(* PLC project PLC Using structs as arrays, CODESYS CODESYS V3.5 SP16, author Toni Kucic *)
(* stored: creationDateTime 2021-02-20T20:12:28.2562031, version 1.0, modificationDateTime 2021-02-20T20:12:09.3479166, organization TK Automation *)
(* A tutorial how to use structs and user derived types as arrays if the PLC IDE/Compiler doesnt allow for arrays. Working with booleans, numbers and user data types is shown in respective POUs that can be run on any PLC that is iec61131-3 compliant. For other data types the process is the same. On top of the examples the project contains struct arrays of 32 elements for each elementary type so the users can start using the functions immediately. If the operator needs different data types the Python generator script can be used. THe python script is located in the same repository as this file. Originally written in CODESYS 3.5. These DTs and POUs can be used under the MIT license. *)

TYPE BOOL32 : STRUCT
  ix00 : BOOL;  (* Index 00 of struct array *)
  ix01 : BOOL;  (* Index 01 of struct array *)
  ix02 : BOOL;  (* Index 02 of struct array *)
  ix03 : BOOL;  (* Index 03 of struct array *)
  ix04 : BOOL;  (* Index 04 of struct array *)
  ix05 : BOOL;  (* Index 05 of struct array *)
  ix06 : BOOL;  (* Index 06 of struct array *)
  ix07 : BOOL;  (* Index 07 of struct array *)
  ix08 : BOOL;  (* Index 08 of struct array *)
  ix09 : BOOL;  (* Index 09 of struct array *)
  ix10 : BOOL;  (* Index 10 of struct array *)
  ix11 : BOOL;  (* Index 11 of struct array *)
  ix12 : BOOL;  (* Index 12 of struct array *)
  ix13 : BOOL;  (* Index 13 of struct array *)
  ix14 : BOOL;  (* Index 14 of struct array *)
  ix15 : BOOL;  (* Index 15 of struct array *)
  ix16 : BOOL;  (* Index 16 of struct array *)
  ix17 : BOOL;  (* Index 17 of struct array *)
  ix18 : BOOL;  (* Index 18 of struct array *)
  ix19 : BOOL;  (* Index 19 of struct array *)
  ix20 : BOOL;  (* Index 20 of struct array *)
  ix21 : BOOL;  (* Index 21 of struct array *)
  ix22 : BOOL;  (* Index 22 of struct array *)
  ix23 : BOOL;  (* Index 23 of struct array *)
  ix24 : BOOL;  (* Index 24 of struct array *)
  ix25 : BOOL;  (* Index 25 of struct array *)
  ix26 : BOOL;  (* Index 26 of struct array *)
  ix27 : BOOL;  (* Index 27 of struct array *)
  ix28 : BOOL;  (* Index 28 of struct array *)
  ix29 : BOOL;  (* Index 29 of struct array *)
  ix30 : BOOL;  (* Index 30 of struct array *)
  ix31 : BOOL;  (* Index 31 of struct array *)
END_STRUCT;
END_TYPE

TYPE BYTE32 : STRUCT
  ix00 : BYTE;  (* Index 00 of struct array *)
  ix01 : BYTE;  (* Index 01 of struct array *)
  ix02 : BYTE;  (* Index 02 of struct array *)
  ix03 : BYTE;  (* Index 03 of struct array *)
  ix04 : BYTE;  (* Index 04 of struct array *)
  ix05 : BYTE;  (* Index 05 of struct array *)
  ix06 : BYTE;  (* Index 06 of struct array *)
  ix07 : BYTE;  (* Index 07 of struct array *)
  ix08 : BYTE;  (* Index 08 of struct array *)
  ix09 : BYTE;  (* Index 09 of struct array *)
  ix10 : BYTE;  (* Index 10 of struct array *)
  ix11 : BYTE;  (* Index 11 of struct array *)
  ix12 : BYTE;  (* Index 12 of struct array *)
  ix13 : BYTE;  (* Index 13 of struct array *)
  ix14 : BYTE;  (* Index 14 of struct array *)
  ix15 : BYTE;  (* Index 15 of struct array *)
  ix16 : BYTE;  (* Index 16 of struct array *)
  ix17 : BYTE;  (* Index 17 of struct array *)
  ix18 : BYTE;  (* Index 18 of struct array *)
  ix19 : BYTE;  (* Index 19 of struct array *)
  ix20 : BYTE;  (* Index 20 of struct array *)
  ix21 : BYTE;  (* Index 21 of struct array *)
  ix22 : BYTE;  (* Index 22 of struct array *)
  ix23 : BYTE;  (* Index 23 of struct array *)
  ix24 : BYTE;  (* Index 24 of struct array *)
  ix25 : BYTE;  (* Index 25 of struct array *)
  ix26 : BYTE;  (* Index 26 of struct array *)
  ix27 : BYTE;  (* Index 27 of struct array *)
  ix28 : BYTE;  (* Index 28 of struct array *)
  ix29 : BYTE;  (* Index 29 of struct array *)
  ix30 : BYTE;  (* Index 30 of struct array *)
  ix31 : BYTE;  (* Index 31 of struct array *)
END_STRUCT;
END_TYPE

TYPE DATE_AND_TIME32 : STRUCT
  ix00 : DT;  (* Index 00 of struct array *)
  ix01 : DT;  (* Index 01 of struct array *)
  ix02 : DT;  (* Index 02 of struct array *)
  ix03 : DT;  (* Index 03 of struct array *)
  ix04 : DT;  (* Index 04 of struct array *)
  ix05 : DT;  (* Index 05 of struct array *)
  ix06 : DT;  (* Index 06 of struct array *)
  ix07 : DT;  (* Index 07 of struct array *)
  ix08 : DT;  (* Index 08 of struct array *)
  ix09 : DT;  (* Index 09 of struct array *)
  ix10 : DT;  (* Index 10 of struct array *)
  ix11 : DT;  (* Index 11 of struct array *)
  ix12 : DT;  (* Index 12 of struct array *)
  ix13 : DT;  (* Index 13 of struct array *)
  ix14 : DT;  (* Index 14 of struct array *)
  ix15 : DT;  (* Index 15 of struct array *)
  ix16 : DT;  (* Index 16 of struct array *)
  ix17 : DT;  (* Index 17 of struct array *)
  ix18 : DT;  (* Index 18 of struct array *)
  ix19 : DT;  (* Index 19 of struct array *)
  ix20 : DT;  (* Index 20 of struct array *)
  ix21 : DT;  (* Index 21 of struct array *)
  ix22 : DT;  (* Index 22 of struct array *)
  ix23 : DT;  (* Index 23 of struct array *)
  ix24 : DT;  (* Index 24 of struct array *)
  ix25 : DT;  (* Index 25 of struct array *)
  ix26 : DT;  (* Index 26 of struct array *)
  ix27 : DT;  (* Index 27 of struct array *)
  ix28 : DT;  (* Index 28 of struct array *)
  ix29 : DT;  (* Index 29 of struct array *)
  ix30 : DT;  (* Index 30 of struct array *)
  ix31 : DT;  (* Index 31 of struct array *)
END_STRUCT;
END_TYPE

TYPE DATE32 : STRUCT
  ix00 : DATE;  (* Index 00 of struct array *)
  ix01 : DATE;  (* Index 01 of struct array *)
  ix02 : DATE;  (* Index 02 of struct array *)
  ix03 : DATE;  (* Index 03 of struct array *)
  ix04 : DATE;  (* Index 04 of struct array *)
  ix05 : DATE;  (* Index 05 of struct array *)
  ix06 : DATE;  (* Index 06 of struct array *)
  ix07 : DATE;  (* Index 07 of struct array *)
  ix08 : DATE;  (* Index 08 of struct array *)
  ix09 : DATE;  (* Index 09 of struct array *)
  ix10 : DATE;  (* Index 10 of struct array *)
  ix11 : DATE;  (* Index 11 of struct array *)
  ix12 : DATE;  (* Index 12 of struct array *)
  ix13 : DATE;  (* Index 13 of struct array *)
  ix14 : DATE;  (* Index 14 of struct array *)
  ix15 : DATE;  (* Index 15 of struct array *)
  ix16 : DATE;  (* Index 16 of struct array *)
  ix17 : DATE;  (* Index 17 of struct array *)
  ix18 : DATE;  (* Index 18 of struct array *)
  ix19 : DATE;  (* Index 19 of struct array *)
  ix20 : DATE;  (* Index 20 of struct array *)
  ix21 : DATE;  (* Index 21 of struct array *)
  ix22 : DATE;  (* Index 22 of struct array *)
  ix23 : DATE;  (* Index 23 of struct array *)
  ix24 : DATE;  (* Index 24 of struct array *)
  ix25 : DATE;  (* Index 25 of struct array *)
  ix26 : DATE;  (* Index 26 of struct array *)
  ix27 : DATE;  (* Index 27 of struct array *)
  ix28 : DATE;  (* Index 28 of struct array *)
  ix29 : DATE;  (* Index 29 of struct array *)
  ix30 : DATE;  (* Index 30 of struct array *)
  ix31 : DATE;  (* Index 31 of struct array *)
END_STRUCT;
END_TYPE

TYPE DINT32 : STRUCT
  ix00 : DINT;  (* Index 00 of struct array *)
  ix01 : DINT;  (* Index 01 of struct array *)
  ix02 : DINT;  (* Index 02 of struct array *)
  ix03 : DINT;  (* Index 03 of struct array *)
  ix04 : DINT;  (* Index 04 of struct array *)
  ix05 : DINT;  (* Index 05 of struct array *)
  ix06 : DINT;  (* Index 06 of struct array *)
  ix07 : DINT;  (* Index 07 of struct array *)
  ix08 : DINT;  (* Index 08 of struct array *)
  ix09 : DINT;  (* Index 09 of struct array *)
  ix10 : DINT;  (* Index 10 of struct array *)
  ix11 : DINT;  (* Index 11 of struct array *)
  ix12 : DINT;  (* Index 12 of struct array *)
  ix13 : DINT;  (* Index 13 of struct array *)
  ix14 : DINT;  (* Index 14 of struct array *)
  ix15 : DINT;  (* Index 15 of struct array *)
  ix16 : DINT;  (* Index 16 of struct array *)
  ix17 : DINT;  (* Index 17 of struct array *)
  ix18 : DINT;  (* Index 18 of struct array *)
  ix19 : DINT;  (* Index 19 of struct array *)
  ix20 : DINT;  (* Index 20 of struct array *)
  ix21 : DINT;  (* Index 21 of struct array *)
  ix22 : DINT;  (* Index 22 of struct array *)
  ix23 : DINT;  (* Index 23 of struct array *)
  ix24 : DINT;  (* Index 24 of struct array *)
  ix25 : DINT;  (* Index 25 of struct array *)
  ix26 : DINT;  (* Index 26 of struct array *)
  ix27 : DINT;  (* Index 27 of struct array *)
  ix28 : DINT;  (* Index 28 of struct array *)
  ix29 : DINT;  (* Index 29 of struct array *)
  ix30 : DINT;  (* Index 30 of struct array *)
  ix31 : DINT;  (* Index 31 of struct array *)
END_STRUCT;
END_TYPE

TYPE DWORD32 : STRUCT
  ix00 : DWORD;  (* Index 00 of struct array *)
  ix01 : DWORD;  (* Index 01 of struct array *)
  ix02 : DWORD;  (* Index 02 of struct array *)
  ix03 : DWORD;  (* Index 03 of struct array *)
  ix04 : DWORD;  (* Index 04 of struct array *)
  ix05 : DWORD;  (* Index 05 of struct array *)
  ix06 : DWORD;  (* Index 06 of struct array *)
  ix07 : DWORD;  (* Index 07 of struct array *)
  ix08 : DWORD;  (* Index 08 of struct array *)
  ix09 : DWORD;  (* Index 09 of struct array *)
  ix10 : DWORD;  (* Index 10 of struct array *)
  ix11 : DWORD;  (* Index 11 of struct array *)
  ix12 : DWORD;  (* Index 12 of struct array *)
  ix13 : DWORD;  (* Index 13 of struct array *)
  ix14 : DWORD;  (* Index 14 of struct array *)
  ix15 : DWORD;  (* Index 15 of struct array *)
  ix16 : DWORD;  (* Index 16 of struct array *)
  ix17 : DWORD;  (* Index 17 of struct array *)
  ix18 : DWORD;  (* Index 18 of struct array *)
  ix19 : DWORD;  (* Index 19 of struct array *)
  ix20 : DWORD;  (* Index 20 of struct array *)
  ix21 : DWORD;  (* Index 21 of struct array *)
  ix22 : DWORD;  (* Index 22 of struct array *)
  ix23 : DWORD;  (* Index 23 of struct array *)
  ix24 : DWORD;  (* Index 24 of struct array *)
  ix25 : DWORD;  (* Index 25 of struct array *)
  ix26 : DWORD;  (* Index 26 of struct array *)
  ix27 : DWORD;  (* Index 27 of struct array *)
  ix28 : DWORD;  (* Index 28 of struct array *)
  ix29 : DWORD;  (* Index 29 of struct array *)
  ix30 : DWORD;  (* Index 30 of struct array *)
  ix31 : DWORD;  (* Index 31 of struct array *)
END_STRUCT;
END_TYPE

TYPE INT32 : STRUCT
  ix00 : INT;  (* Index 00 of struct array *)
  ix01 : INT;  (* Index 01 of struct array *)
  ix02 : INT;  (* Index 02 of struct array *)
  ix03 : INT;  (* Index 03 of struct array *)
  ix04 : INT;  (* Index 04 of struct array *)
  ix05 : INT;  (* Index 05 of struct array *)
  ix06 : INT;  (* Index 06 of struct array *)
  ix07 : INT;  (* Index 07 of struct array *)
  ix08 : INT;  (* Index 08 of struct array *)
  ix09 : INT;  (* Index 09 of struct array *)
  ix10 : INT;  (* Index 10 of struct array *)
  ix11 : INT;  (* Index 11 of struct array *)
  ix12 : INT;  (* Index 12 of struct array *)
  ix13 : INT;  (* Index 13 of struct array *)
  ix14 : INT;  (* Index 14 of struct array *)
  ix15 : INT;  (* Index 15 of struct array *)
  ix16 : INT;  (* Index 16 of struct array *)
  ix17 : INT;  (* Index 17 of struct array *)
  ix18 : INT;  (* Index 18 of struct array *)
  ix19 : INT;  (* Index 19 of struct array *)
  ix20 : INT;  (* Index 20 of struct array *)
  ix21 : INT;  (* Index 21 of struct array *)
  ix22 : INT;  (* Index 22 of struct array *)
  ix23 : INT;  (* Index 23 of struct array *)
  ix24 : INT;  (* Index 24 of struct array *)
  ix25 : INT;  (* Index 25 of struct array *)
  ix26 : INT;  (* Index 26 of struct array *)
  ix27 : INT;  (* Index 27 of struct array *)
  ix28 : INT;  (* Index 28 of struct array *)
  ix29 : INT;  (* Index 29 of struct array *)
  ix30 : INT;  (* Index 30 of struct array *)
  ix31 : INT;  (* Index 31 of struct array *)
END_STRUCT;
END_TYPE

TYPE LDATE_AND_TIME32 : STRUCT
  ix00 : LDATE_AND_TIME;  (* Index 00 of struct array *)
  ix01 : LDATE_AND_TIME;  (* Index 01 of struct array *)
  ix02 : LDATE_AND_TIME;  (* Index 02 of struct array *)
  ix03 : LDATE_AND_TIME;  (* Index 03 of struct array *)
  ix04 : LDATE_AND_TIME;  (* Index 04 of struct array *)
  ix05 : LDATE_AND_TIME;  (* Index 05 of struct array *)
  ix06 : LDATE_AND_TIME;  (* Index 06 of struct array *)
  ix07 : LDATE_AND_TIME;  (* Index 07 of struct array *)
  ix08 : LDATE_AND_TIME;  (* Index 08 of struct array *)
  ix09 : LDATE_AND_TIME;  (* Index 09 of struct array *)
  ix10 : LDATE_AND_TIME;  (* Index 10 of struct array *)
  ix11 : LDATE_AND_TIME;  (* Index 11 of struct array *)
  ix12 : LDATE_AND_TIME;  (* Index 12 of struct array *)
  ix13 : LDATE_AND_TIME;  (* Index 13 of struct array *)
  ix14 : LDATE_AND_TIME;  (* Index 14 of struct array *)
  ix15 : LDATE_AND_TIME;  (* Index 15 of struct array *)
  ix16 : LDATE_AND_TIME;  (* Index 16 of struct array *)
  ix17 : LDATE_AND_TIME;  (* Index 17 of struct array *)
  ix18 : LDATE_AND_TIME;  (* Index 18 of struct array *)
  ix19 : LDATE_AND_TIME;  (* Index 19 of struct array *)
  ix20 : LDATE_AND_TIME;  (* Index 20 of struct array *)
  ix21 : LDATE_AND_TIME;  (* Index 21 of struct array *)
  ix22 : LDATE_AND_TIME;  (* Index 22 of struct array *)
  ix23 : LDATE_AND_TIME;  (* Index 23 of struct array *)
  ix24 : LDATE_AND_TIME;  (* Index 24 of struct array *)
  ix25 : LDATE_AND_TIME;  (* Index 25 of struct array *)
  ix26 : LDATE_AND_TIME;  (* Index 26 of struct array *)
  ix27 : LDATE_AND_TIME;  (* Index 27 of struct array *)
  ix28 : LDATE_AND_TIME;  (* Index 28 of struct array *)
  ix29 : LDATE_AND_TIME;  (* Index 29 of struct array *)
  ix30 : LDATE_AND_TIME;  (* Index 30 of struct array *)
  ix31 : LDATE_AND_TIME;  (* Index 31 of struct array *)
END_STRUCT;
END_TYPE

TYPE LDATE32 : STRUCT
  ix00 : LDATE;  (* Index 00 of struct array *)
  ix01 : LDATE;  (* Index 01 of struct array *)
  ix02 : LDATE;  (* Index 02 of struct array *)
  ix03 : LDATE;  (* Index 03 of struct array *)
  ix04 : LDATE;  (* Index 04 of struct array *)
  ix05 : LDATE;  (* Index 05 of struct array *)
  ix06 : LDATE;  (* Index 06 of struct array *)
  ix07 : LDATE;  (* Index 07 of struct array *)
  ix08 : LDATE;  (* Index 08 of struct array *)
  ix09 : LDATE;  (* Index 09 of struct array *)
  ix10 : LDATE;  (* Index 10 of struct array *)
  ix11 : LDATE;  (* Index 11 of struct array *)
  ix12 : LDATE;  (* Index 12 of struct array *)
  ix13 : LDATE;  (* Index 13 of struct array *)
  ix14 : LDATE;  (* Index 14 of struct array *)
  ix15 : LDATE;  (* Index 15 of struct array *)
  ix16 : LDATE;  (* Index 16 of struct array *)
  ix17 : LDATE;  (* Index 17 of struct array *)
  ix18 : LDATE;  (* Index 18 of struct array *)
  ix19 : LDATE;  (* Index 19 of struct array *)
  ix20 : LDATE;  (* Index 20 of struct array *)
  ix21 : LDATE;  (* Index 21 of struct array *)
  ix22 : LDATE;  (* Index 22 of struct array *)
  ix23 : LDATE;  (* Index 23 of struct array *)
  ix24 : LDATE;  (* Index 24 of struct array *)
  ix25 : LDATE;  (* Index 25 of struct array *)
  ix26 : LDATE;  (* Index 26 of struct array *)
  ix27 : LDATE;  (* Index 27 of struct array *)
  ix28 : LDATE;  (* Index 28 of struct array *)
  ix29 : LDATE;  (* Index 29 of struct array *)
  ix30 : LDATE;  (* Index 30 of struct array *)
  ix31 : LDATE;  (* Index 31 of struct array *)
END_STRUCT;
END_TYPE

TYPE LINT32 : STRUCT
  ix00 : LINT;  (* Index 00 of struct array *)
  ix01 : LINT;  (* Index 01 of struct array *)
  ix02 : LINT;  (* Index 02 of struct array *)
  ix03 : LINT;  (* Index 03 of struct array *)
  ix04 : LINT;  (* Index 04 of struct array *)
  ix05 : LINT;  (* Index 05 of struct array *)
  ix06 : LINT;  (* Index 06 of struct array *)
  ix07 : LINT;  (* Index 07 of struct array *)
  ix08 : LINT;  (* Index 08 of struct array *)
  ix09 : LINT;  (* Index 09 of struct array *)
  ix10 : LINT;  (* Index 10 of struct array *)
  ix11 : LINT;  (* Index 11 of struct array *)
  ix12 : LINT;  (* Index 12 of struct array *)
  ix13 : LINT;  (* Index 13 of struct array *)
  ix14 : LINT;  (* Index 14 of struct array *)
  ix15 : LINT;  (* Index 15 of struct array *)
  ix16 : LINT;  (* Index 16 of struct array *)
  ix17 : LINT;  (* Index 17 of struct array *)
  ix18 : LINT;  (* Index 18 of struct array *)
  ix19 : LINT;  (* Index 19 of struct array *)
  ix20 : LINT;  (* Index 20 of struct array *)
  ix21 : LINT;  (* Index 21 of struct array *)
  ix22 : LINT;  (* Index 22 of struct array *)
  ix23 : LINT;  (* Index 23 of struct array *)
  ix24 : LINT;  (* Index 24 of struct array *)
  ix25 : LINT;  (* Index 25 of struct array *)
  ix26 : LINT;  (* Index 26 of struct array *)
  ix27 : LINT;  (* Index 27 of struct array *)
  ix28 : LINT;  (* Index 28 of struct array *)
  ix29 : LINT;  (* Index 29 of struct array *)
  ix30 : LINT;  (* Index 30 of struct array *)
  ix31 : LINT;  (* Index 31 of struct array *)
END_STRUCT;
END_TYPE

TYPE LREAL32 : STRUCT
  ix00 : LREAL;  (* Index 00 of struct array *)
  ix01 : LREAL;  (* Index 01 of struct array *)
  ix02 : LREAL;  (* Index 02 of struct array *)
  ix03 : LREAL;  (* Index 03 of struct array *)
  ix04 : LREAL;  (* Index 04 of struct array *)
  ix05 : LREAL;  (* Index 05 of struct array *)
  ix06 : LREAL;  (* Index 06 of struct array *)
  ix07 : LREAL;  (* Index 07 of struct array *)
  ix08 : LREAL;  (* Index 08 of struct array *)
  ix09 : LREAL;  (* Index 09 of struct array *)
  ix10 : LREAL;  (* Index 10 of struct array *)
  ix11 : LREAL;  (* Index 11 of struct array *)
  ix12 : LREAL;  (* Index 12 of struct array *)
  ix13 : LREAL;  (* Index 13 of struct array *)
  ix14 : LREAL;  (* Index 14 of struct array *)
  ix15 : LREAL;  (* Index 15 of struct array *)
  ix16 : LREAL;  (* Index 16 of struct array *)
  ix17 : LREAL;  (* Index 17 of struct array *)
  ix18 : LREAL;  (* Index 18 of struct array *)
  ix19 : LREAL;  (* Index 19 of struct array *)
  ix20 : LREAL;  (* Index 20 of struct array *)
  ix21 : LREAL;  (* Index 21 of struct array *)
  ix22 : LREAL;  (* Index 22 of struct array *)
  ix23 : LREAL;  (* Index 23 of struct array *)
  ix24 : LREAL;  (* Index 24 of struct array *)
  ix25 : LREAL;  (* Index 25 of struct array *)
  ix26 : LREAL;  (* Index 26 of struct array *)
  ix27 : LREAL;  (* Index 27 of struct array *)
  ix28 : LREAL;  (* Index 28 of struct array *)
  ix29 : LREAL;  (* Index 29 of struct array *)
  ix30 : LREAL;  (* Index 30 of struct array *)
  ix31 : LREAL;  (* Index 31 of struct array *)
END_STRUCT;
END_TYPE

TYPE LTIME_OF_DAY32 : STRUCT
  ix00 : LTIME_OF_DAY;  (* Index 00 of struct array *)
  ix01 : LTIME_OF_DAY;  (* Index 01 of struct array *)
  ix02 : LTIME_OF_DAY;  (* Index 02 of struct array *)
  ix03 : LTIME_OF_DAY;  (* Index 03 of struct array *)
  ix04 : LTIME_OF_DAY;  (* Index 04 of struct array *)
  ix05 : LTIME_OF_DAY;  (* Index 05 of struct array *)
  ix06 : LTIME_OF_DAY;  (* Index 06 of struct array *)
  ix07 : LTIME_OF_DAY;  (* Index 07 of struct array *)
  ix08 : LTIME_OF_DAY;  (* Index 08 of struct array *)
  ix09 : LTIME_OF_DAY;  (* Index 09 of struct array *)
  ix10 : LTIME_OF_DAY;  (* Index 10 of struct array *)
  ix11 : LTIME_OF_DAY;  (* Index 11 of struct array *)
  ix12 : LTIME_OF_DAY;  (* Index 12 of struct array *)
  ix13 : LTIME_OF_DAY;  (* Index 13 of struct array *)
  ix14 : LTIME_OF_DAY;  (* Index 14 of struct array *)
  ix15 : LTIME_OF_DAY;  (* Index 15 of struct array *)
  ix16 : LTIME_OF_DAY;  (* Index 16 of struct array *)
  ix17 : LTIME_OF_DAY;  (* Index 17 of struct array *)
  ix18 : LTIME_OF_DAY;  (* Index 18 of struct array *)
  ix19 : LTIME_OF_DAY;  (* Index 19 of struct array *)
  ix20 : LTIME_OF_DAY;  (* Index 20 of struct array *)
  ix21 : LTIME_OF_DAY;  (* Index 21 of struct array *)
  ix22 : LTIME_OF_DAY;  (* Index 22 of struct array *)
  ix23 : LTIME_OF_DAY;  (* Index 23 of struct array *)
  ix24 : LTIME_OF_DAY;  (* Index 24 of struct array *)
  ix25 : LTIME_OF_DAY;  (* Index 25 of struct array *)
  ix26 : LTIME_OF_DAY;  (* Index 26 of struct array *)
  ix27 : LTIME_OF_DAY;  (* Index 27 of struct array *)
  ix28 : LTIME_OF_DAY;  (* Index 28 of struct array *)
  ix29 : LTIME_OF_DAY;  (* Index 29 of struct array *)
  ix30 : LTIME_OF_DAY;  (* Index 30 of struct array *)
  ix31 : LTIME_OF_DAY;  (* Index 31 of struct array *)
END_STRUCT;
END_TYPE

TYPE LTIME32 : STRUCT
  ix00 : LTIME;  (* Index 00 of struct array *)
  ix01 : LTIME;  (* Index 01 of struct array *)
  ix02 : LTIME;  (* Index 02 of struct array *)
  ix03 : LTIME;  (* Index 03 of struct array *)
  ix04 : LTIME;  (* Index 04 of struct array *)
  ix05 : LTIME;  (* Index 05 of struct array *)
  ix06 : LTIME;  (* Index 06 of struct array *)
  ix07 : LTIME;  (* Index 07 of struct array *)
  ix08 : LTIME;  (* Index 08 of struct array *)
  ix09 : LTIME;  (* Index 09 of struct array *)
  ix10 : LTIME;  (* Index 10 of struct array *)
  ix11 : LTIME;  (* Index 11 of struct array *)
  ix12 : LTIME;  (* Index 12 of struct array *)
  ix13 : LTIME;  (* Index 13 of struct array *)
  ix14 : LTIME;  (* Index 14 of struct array *)
  ix15 : LTIME;  (* Index 15 of struct array *)
  ix16 : LTIME;  (* Index 16 of struct array *)
  ix17 : LTIME;  (* Index 17 of struct array *)
  ix18 : LTIME;  (* Index 18 of struct array *)
  ix19 : LTIME;  (* Index 19 of struct array *)
  ix20 : LTIME;  (* Index 20 of struct array *)
  ix21 : LTIME;  (* Index 21 of struct array *)
  ix22 : LTIME;  (* Index 22 of struct array *)
  ix23 : LTIME;  (* Index 23 of struct array *)
  ix24 : LTIME;  (* Index 24 of struct array *)
  ix25 : LTIME;  (* Index 25 of struct array *)
  ix26 : LTIME;  (* Index 26 of struct array *)
  ix27 : LTIME;  (* Index 27 of struct array *)
  ix28 : LTIME;  (* Index 28 of struct array *)
  ix29 : LTIME;  (* Index 29 of struct array *)
  ix30 : LTIME;  (* Index 30 of struct array *)
  ix31 : LTIME;  (* Index 31 of struct array *)
END_STRUCT;
END_TYPE

TYPE LWORD32 : STRUCT
  ix00 : LWORD;  (* Index 00 of struct array *)
  ix01 : LWORD;  (* Index 01 of struct array *)
  ix02 : LWORD;  (* Index 02 of struct array *)
  ix03 : LWORD;  (* Index 03 of struct array *)
  ix04 : LWORD;  (* Index 04 of struct array *)
  ix05 : LWORD;  (* Index 05 of struct array *)
  ix06 : LWORD;  (* Index 06 of struct array *)
  ix07 : LWORD;  (* Index 07 of struct array *)
  ix08 : LWORD;  (* Index 08 of struct array *)
  ix09 : LWORD;  (* Index 09 of struct array *)
  ix10 : LWORD;  (* Index 10 of struct array *)
  ix11 : LWORD;  (* Index 11 of struct array *)
  ix12 : LWORD;  (* Index 12 of struct array *)
  ix13 : LWORD;  (* Index 13 of struct array *)
  ix14 : LWORD;  (* Index 14 of struct array *)
  ix15 : LWORD;  (* Index 15 of struct array *)
  ix16 : LWORD;  (* Index 16 of struct array *)
  ix17 : LWORD;  (* Index 17 of struct array *)
  ix18 : LWORD;  (* Index 18 of struct array *)
  ix19 : LWORD;  (* Index 19 of struct array *)
  ix20 : LWORD;  (* Index 20 of struct array *)
  ix21 : LWORD;  (* Index 21 of struct array *)
  ix22 : LWORD;  (* Index 22 of struct array *)
  ix23 : LWORD;  (* Index 23 of struct array *)
  ix24 : LWORD;  (* Index 24 of struct array *)
  ix25 : LWORD;  (* Index 25 of struct array *)
  ix26 : LWORD;  (* Index 26 of struct array *)
  ix27 : LWORD;  (* Index 27 of struct array *)
  ix28 : LWORD;  (* Index 28 of struct array *)
  ix29 : LWORD;  (* Index 29 of struct array *)
  ix30 : LWORD;  (* Index 30 of struct array *)
  ix31 : LWORD;  (* Index 31 of struct array *)
END_STRUCT;
END_TYPE

TYPE REAL32 : STRUCT
  ix00 : REAL;  (* Index 00 of struct array *)
  ix01 : REAL;  (* Index 01 of struct array *)
  ix02 : REAL;  (* Index 02 of struct array *)
  ix03 : REAL;  (* Index 03 of struct array *)
  ix04 : REAL;  (* Index 04 of struct array *)
  ix05 : REAL;  (* Index 05 of struct array *)
  ix06 : REAL;  (* Index 06 of struct array *)
  ix07 : REAL;  (* Index 07 of struct array *)
  ix08 : REAL;  (* Index 08 of struct array *)
  ix09 : REAL;  (* Index 09 of struct array *)
  ix10 : REAL;  (* Index 10 of struct array *)
  ix11 : REAL;  (* Index 11 of struct array *)
  ix12 : REAL;  (* Index 12 of struct array *)
  ix13 : REAL;  (* Index 13 of struct array *)
  ix14 : REAL;  (* Index 14 of struct array *)
  ix15 : REAL;  (* Index 15 of struct array *)
  ix16 : REAL;  (* Index 16 of struct array *)
  ix17 : REAL;  (* Index 17 of struct array *)
  ix18 : REAL;  (* Index 18 of struct array *)
  ix19 : REAL;  (* Index 19 of struct array *)
  ix20 : REAL;  (* Index 20 of struct array *)
  ix21 : REAL;  (* Index 21 of struct array *)
  ix22 : REAL;  (* Index 22 of struct array *)
  ix23 : REAL;  (* Index 23 of struct array *)
  ix24 : REAL;  (* Index 24 of struct array *)
  ix25 : REAL;  (* Index 25 of struct array *)
  ix26 : REAL;  (* Index 26 of struct array *)
  ix27 : REAL;  (* Index 27 of struct array *)
  ix28 : REAL;  (* Index 28 of struct array *)
  ix29 : REAL;  (* Index 29 of struct array *)
  ix30 : REAL;  (* Index 30 of struct array *)
  ix31 : REAL;  (* Index 31 of struct array *)
END_STRUCT;
END_TYPE

TYPE SINT32 : STRUCT
  ix00 : SINT;  (* Index 00 of struct array *)
  ix01 : SINT;  (* Index 01 of struct array *)
  ix02 : SINT;  (* Index 02 of struct array *)
  ix03 : SINT;  (* Index 03 of struct array *)
  ix04 : SINT;  (* Index 04 of struct array *)
  ix05 : SINT;  (* Index 05 of struct array *)
  ix06 : SINT;  (* Index 06 of struct array *)
  ix07 : SINT;  (* Index 07 of struct array *)
  ix08 : SINT;  (* Index 08 of struct array *)
  ix09 : SINT;  (* Index 09 of struct array *)
  ix10 : SINT;  (* Index 10 of struct array *)
  ix11 : SINT;  (* Index 11 of struct array *)
  ix12 : SINT;  (* Index 12 of struct array *)
  ix13 : SINT;  (* Index 13 of struct array *)
  ix14 : SINT;  (* Index 14 of struct array *)
  ix15 : SINT;  (* Index 15 of struct array *)
  ix16 : SINT;  (* Index 16 of struct array *)
  ix17 : SINT;  (* Index 17 of struct array *)
  ix18 : SINT;  (* Index 18 of struct array *)
  ix19 : SINT;  (* Index 19 of struct array *)
  ix20 : SINT;  (* Index 20 of struct array *)
  ix21 : SINT;  (* Index 21 of struct array *)
  ix22 : SINT;  (* Index 22 of struct array *)
  ix23 : SINT;  (* Index 23 of struct array *)
  ix24 : SINT;  (* Index 24 of struct array *)
  ix25 : SINT;  (* Index 25 of struct array *)
  ix26 : SINT;  (* Index 26 of struct array *)
  ix27 : SINT;  (* Index 27 of struct array *)
  ix28 : SINT;  (* Index 28 of struct array *)
  ix29 : SINT;  (* Index 29 of struct array *)
  ix30 : SINT;  (* Index 30 of struct array *)
  ix31 : SINT;  (* Index 31 of struct array *)
END_STRUCT;
END_TYPE

TYPE STRING32 : STRUCT
  ix00 : STRING;  (* Index 00 of struct array *)
  ix01 : STRING;  (* Index 01 of struct array *)
  ix02 : STRING;  (* Index 02 of struct array *)
  ix03 : STRING;  (* Index 03 of struct array *)
  ix04 : STRING;  (* Index 04 of struct array *)
  ix05 : STRING;  (* Index 05 of struct array *)
  ix06 : STRING;  (* Index 06 of struct array *)
  ix07 : STRING;  (* Index 07 of struct array *)
  ix08 : STRING;  (* Index 08 of struct array *)
  ix09 : STRING;  (* Index 09 of struct array *)
  ix10 : STRING;  (* Index 10 of struct array *)
  ix11 : STRING;  (* Index 11 of struct array *)
  ix12 : STRING;  (* Index 12 of struct array *)
  ix13 : STRING;  (* Index 13 of struct array *)
  ix14 : STRING;  (* Index 14 of struct array *)
  ix15 : STRING;  (* Index 15 of struct array *)
  ix16 : STRING;  (* Index 16 of struct array *)
  ix17 : STRING;  (* Index 17 of struct array *)
  ix18 : STRING;  (* Index 18 of struct array *)
  ix19 : STRING;  (* Index 19 of struct array *)
  ix20 : STRING;  (* Index 20 of struct array *)
  ix21 : STRING;  (* Index 21 of struct array *)
  ix22 : STRING;  (* Index 22 of struct array *)
  ix23 : STRING;  (* Index 23 of struct array *)
  ix24 : STRING;  (* Index 24 of struct array *)
  ix25 : STRING;  (* Index 25 of struct array *)
  ix26 : STRING;  (* Index 26 of struct array *)
  ix27 : STRING;  (* Index 27 of struct array *)
  ix28 : STRING;  (* Index 28 of struct array *)
  ix29 : STRING;  (* Index 29 of struct array *)
  ix30 : STRING;  (* Index 30 of struct array *)
  ix31 : STRING;  (* Index 31 of struct array *)
END_STRUCT;
END_TYPE

TYPE TIME_OF_DAY32 : STRUCT
  ix00 : TOD;  (* Index 00 of struct array *)
  ix01 : TOD;  (* Index 01 of struct array *)
  ix02 : TOD;  (* Index 02 of struct array *)
  ix03 : TOD;  (* Index 03 of struct array *)
  ix04 : TOD;  (* Index 04 of struct array *)
  ix05 : TOD;  (* Index 05 of struct array *)
  ix06 : TOD;  (* Index 06 of struct array *)
  ix07 : TOD;  (* Index 07 of struct array *)
  ix08 : TOD;  (* Index 08 of struct array *)
  ix09 : TOD;  (* Index 09 of struct array *)
  ix10 : TOD;  (* Index 10 of struct array *)
  ix11 : TOD;  (* Index 11 of struct array *)
  ix12 : TOD;  (* Index 12 of struct array *)
  ix13 : TOD;  (* Index 13 of struct array *)
  ix14 : TOD;  (* Index 14 of struct array *)
  ix15 : TOD;  (* Index 15 of struct array *)
  ix16 : TOD;  (* Index 16 of struct array *)
  ix17 : TOD;  (* Index 17 of struct array *)
  ix18 : TOD;  (* Index 18 of struct array *)
  ix19 : TOD;  (* Index 19 of struct array *)
  ix20 : TOD;  (* Index 20 of struct array *)
  ix21 : TOD;  (* Index 21 of struct array *)
  ix22 : TOD;  (* Index 22 of struct array *)
  ix23 : TOD;  (* Index 23 of struct array *)
  ix24 : TOD;  (* Index 24 of struct array *)
  ix25 : TOD;  (* Index 25 of struct array *)
  ix26 : TOD;  (* Index 26 of struct array *)
  ix27 : TOD;  (* Index 27 of struct array *)
  ix28 : TOD;  (* Index 28 of struct array *)
  ix29 : TOD;  (* Index 29 of struct array *)
  ix30 : TOD;  (* Index 30 of struct array *)
  ix31 : TOD;  (* Index 31 of struct array *)
END_STRUCT;
END_TYPE

TYPE TIME32 : STRUCT
  ix00 : TIME;  (* Index 00 of struct array *)
  ix01 : TIME;  (* Index 01 of struct array *)
  ix02 : TIME;  (* Index 02 of struct array *)
  ix03 : TIME;  (* Index 03 of struct array *)
  ix04 : TIME;  (* Index 04 of struct array *)
  ix05 : TIME;  (* Index 05 of struct array *)
  ix06 : TIME;  (* Index 06 of struct array *)
  ix07 : TIME;  (* Index 07 of struct array *)
  ix08 : TIME;  (* Index 08 of struct array *)
  ix09 : TIME;  (* Index 09 of struct array *)
  ix10 : TIME;  (* Index 10 of struct array *)
  ix11 : TIME;  (* Index 11 of struct array *)
  ix12 : TIME;  (* Index 12 of struct array *)
  ix13 : TIME;  (* Index 13 of struct array *)
  ix14 : TIME;  (* Index 14 of struct array *)
  ix15 : TIME;  (* Index 15 of struct array *)
  ix16 : TIME;  (* Index 16 of struct array *)
  ix17 : TIME;  (* Index 17 of struct array *)
  ix18 : TIME;  (* Index 18 of struct array *)
  ix19 : TIME;  (* Index 19 of struct array *)
  ix20 : TIME;  (* Index 20 of struct array *)
  ix21 : TIME;  (* Index 21 of struct array *)
  ix22 : TIME;  (* Index 22 of struct array *)
  ix23 : TIME;  (* Index 23 of struct array *)
  ix24 : TIME;  (* Index 24 of struct array *)
  ix25 : TIME;  (* Index 25 of struct array *)
  ix26 : TIME;  (* Index 26 of struct array *)
  ix27 : TIME;  (* Index 27 of struct array *)
  ix28 : TIME;  (* Index 28 of struct array *)
  ix29 : TIME;  (* Index 29 of struct array *)
  ix30 : TIME;  (* Index 30 of struct array *)
  ix31 : TIME;  (* Index 31 of struct array *)
END_STRUCT;
END_TYPE

TYPE UDINT32 : STRUCT
  ix00 : UDINT;  (* Index 00 of struct array *)
  ix01 : UDINT;  (* Index 01 of struct array *)
  ix02 : UDINT;  (* Index 02 of struct array *)
  ix03 : UDINT;  (* Index 03 of struct array *)
  ix04 : UDINT;  (* Index 04 of struct array *)
  ix05 : UDINT;  (* Index 05 of struct array *)
  ix06 : UDINT;  (* Index 06 of struct array *)
  ix07 : UDINT;  (* Index 07 of struct array *)
  ix08 : UDINT;  (* Index 08 of struct array *)
  ix09 : UDINT;  (* Index 09 of struct array *)
  ix10 : UDINT;  (* Index 10 of struct array *)
  ix11 : UDINT;  (* Index 11 of struct array *)
  ix12 : UDINT;  (* Index 12 of struct array *)
  ix13 : UDINT;  (* Index 13 of struct array *)
  ix14 : UDINT;  (* Index 14 of struct array *)
  ix15 : UDINT;  (* Index 15 of struct array *)
  ix16 : UDINT;  (* Index 16 of struct array *)
  ix17 : UDINT;  (* Index 17 of struct array *)
  ix18 : UDINT;  (* Index 18 of struct array *)
  ix19 : UDINT;  (* Index 19 of struct array *)
  ix20 : UDINT;  (* Index 20 of struct array *)
  ix21 : UDINT;  (* Index 21 of struct array *)
  ix22 : UDINT;  (* Index 22 of struct array *)
  ix23 : UDINT;  (* Index 23 of struct array *)
  ix24 : UDINT;  (* Index 24 of struct array *)
  ix25 : UDINT;  (* Index 25 of struct array *)
  ix26 : UDINT;  (* Index 26 of struct array *)
  ix27 : UDINT;  (* Index 27 of struct array *)
  ix28 : UDINT;  (* Index 28 of struct array *)
  ix29 : UDINT;  (* Index 29 of struct array *)
  ix30 : UDINT;  (* Index 30 of struct array *)
  ix31 : UDINT;  (* Index 31 of struct array *)
END_STRUCT;
END_TYPE

TYPE UDT_Cmd : STRUCT
  StartCmd : BOOL;  (* Start command to the device *)
  StopCmd : BOOL;  (* Stop command to the device *)
  ResetCmd : BOOL;  (* Reset command for the device *)
  Ref : REAL;  (* Reference for the device to follow *)
END_STRUCT;
END_TYPE

TYPE UDT_Cmd32 : STRUCT
  udt00 : UDT_Cmd;  (* User data type array index 0 *)
  udt01 : UDT_Cmd;  (* User data type array index 1 *)
  udt02 : UDT_Cmd;  (* User data type array index 2 *)
  udt03 : UDT_Cmd;  (* User data type array index 3 *)
  udt04 : UDT_Cmd;  (* User data type array index 4 *)
  udt05 : UDT_Cmd;  (* User data type array index 5 *)
  udt06 : UDT_Cmd;  (* User data type array index 6 *)
  udt07 : UDT_Cmd;  (* User data type array index 7 *)
  udt08 : UDT_Cmd;  (* User data type array index 8 *)
  udt09 : UDT_Cmd;  (* User data type array index 9 *)
  udt10 : UDT_Cmd;  (* User data type array index 10 *)
  udt11 : UDT_Cmd;  (* User data type array index 11 *)
  udt12 : UDT_Cmd;  (* User data type array index 12 *)
  udt13 : UDT_Cmd;  (* User data type array index 13 *)
  udt14 : UDT_Cmd;  (* User data type array index 14 *)
  udt15 : UDT_Cmd;  (* User data type array index 15 *)
  udt16 : UDT_Cmd;  (* User data type array index 16 *)
  udt17 : UDT_Cmd;  (* User data type array index 17 *)
  udt18 : UDT_Cmd;  (* User data type array index 18 *)
  udt19 : UDT_Cmd;  (* User data type array index 19 *)
  udt20 : UDT_Cmd;  (* User data type array index 20 *)
  udt21 : UDT_Cmd;  (* User data type array index 21 *)
  udt22 : UDT_Cmd;  (* User data type array index 22 *)
  udt23 : UDT_Cmd;  (* User data type array index 23 *)
  udt24 : UDT_Cmd;  (* User data type array index 24 *)
  udt25 : UDT_Cmd;  (* User data type array index 25 *)
  udt26 : UDT_Cmd;  (* User data type array index 26 *)
  udt27 : UDT_Cmd;  (* User data type array index 27 *)
  udt28 : UDT_Cmd;  (* User data type array index 28 *)
  udt29 : UDT_Cmd;  (* User data type array index 29 *)
  udt30 : UDT_Cmd;  (* User data type array index 30 *)
  udt31 : UDT_Cmd;  (* User data type array index 31 *)
END_STRUCT;
END_TYPE

TYPE UDT_Status : STRUCT
  Running : BOOL;  (* Device is running *)
  ResetRequired : BOOL;  (* Device needs a reset *)
  RefActual : REAL;  (* Devices used reference *)
END_STRUCT;
END_TYPE

TYPE UDT_Status32 : STRUCT
  udt00 : UDT_Status;  (* User data type array index 0 *)
  udt01 : UDT_Status;  (* User data type array index 1 *)
  udt02 : UDT_Status;  (* User data type array index 2 *)
  udt03 : UDT_Status;  (* User data type array index 3 *)
  udt04 : UDT_Status;  (* User data type array index 4 *)
  udt05 : UDT_Status;  (* User data type array index 5 *)
  udt06 : UDT_Status;  (* User data type array index 6 *)
  udt07 : UDT_Status;  (* User data type array index 7 *)
  udt08 : UDT_Status;  (* User data type array index 8 *)
  udt09 : UDT_Status;  (* User data type array index 9 *)
  udt10 : UDT_Status;  (* User data type array index 10 *)
  udt11 : UDT_Status;  (* User data type array index 11 *)
  udt12 : UDT_Status;  (* User data type array index 12 *)
  udt13 : UDT_Status;  (* User data type array index 13 *)
  udt14 : UDT_Status;  (* User data type array index 14 *)
  udt15 : UDT_Status;  (* User data type array index 15 *)
  udt16 : UDT_Status;  (* User data type array index 16 *)
  udt17 : UDT_Status;  (* User data type array index 17 *)
  udt18 : UDT_Status;  (* User data type array index 18 *)
  udt19 : UDT_Status;  (* User data type array index 19 *)
  udt20 : UDT_Status;  (* User data type array index 20 *)
  udt21 : UDT_Status;  (* User data type array index 21 *)
  udt22 : UDT_Status;  (* User data type array index 22 *)
  udt23 : UDT_Status;  (* User data type array index 23 *)
  udt24 : UDT_Status;  (* User data type array index 24 *)
  udt25 : UDT_Status;  (* User data type array index 25 *)
  udt26 : UDT_Status;  (* User data type array index 26 *)
  udt27 : UDT_Status;  (* User data type array index 27 *)
  udt28 : UDT_Status;  (* User data type array index 28 *)
  udt29 : UDT_Status;  (* User data type array index 29 *)
  udt30 : UDT_Status;  (* User data type array index 30 *)
  udt31 : UDT_Status;  (* User data type array index 31 *)
END_STRUCT;
END_TYPE

TYPE UINT32 : STRUCT
  ix00 : UINT;  (* Index 00 of struct array *)
  ix01 : UINT;  (* Index 01 of struct array *)
  ix02 : UINT;  (* Index 02 of struct array *)
  ix03 : UINT;  (* Index 03 of struct array *)
  ix04 : UINT;  (* Index 04 of struct array *)
  ix05 : UINT;  (* Index 05 of struct array *)
  ix06 : UINT;  (* Index 06 of struct array *)
  ix07 : UINT;  (* Index 07 of struct array *)
  ix08 : UINT;  (* Index 08 of struct array *)
  ix09 : UINT;  (* Index 09 of struct array *)
  ix10 : UINT;  (* Index 10 of struct array *)
  ix11 : UINT;  (* Index 11 of struct array *)
  ix12 : UINT;  (* Index 12 of struct array *)
  ix13 : UINT;  (* Index 13 of struct array *)
  ix14 : UINT;  (* Index 14 of struct array *)
  ix15 : UINT;  (* Index 15 of struct array *)
  ix16 : UINT;  (* Index 16 of struct array *)
  ix17 : UINT;  (* Index 17 of struct array *)
  ix18 : UINT;  (* Index 18 of struct array *)
  ix19 : UINT;  (* Index 19 of struct array *)
  ix20 : UINT;  (* Index 20 of struct array *)
  ix21 : UINT;  (* Index 21 of struct array *)
  ix22 : UINT;  (* Index 22 of struct array *)
  ix23 : UINT;  (* Index 23 of struct array *)
  ix24 : UINT;  (* Index 24 of struct array *)
  ix25 : UINT;  (* Index 25 of struct array *)
  ix26 : UINT;  (* Index 26 of struct array *)
  ix27 : UINT;  (* Index 27 of struct array *)
  ix28 : UINT;  (* Index 28 of struct array *)
  ix29 : UINT;  (* Index 29 of struct array *)
  ix30 : UINT;  (* Index 30 of struct array *)
  ix31 : UINT;  (* Index 31 of struct array *)
END_STRUCT;
END_TYPE

TYPE ULINT32 : STRUCT
  ix00 : ULINT;  (* Index 00 of struct array *)
  ix01 : ULINT;  (* Index 01 of struct array *)
  ix02 : ULINT;  (* Index 02 of struct array *)
  ix03 : ULINT;  (* Index 03 of struct array *)
  ix04 : ULINT;  (* Index 04 of struct array *)
  ix05 : ULINT;  (* Index 05 of struct array *)
  ix06 : ULINT;  (* Index 06 of struct array *)
  ix07 : ULINT;  (* Index 07 of struct array *)
  ix08 : ULINT;  (* Index 08 of struct array *)
  ix09 : ULINT;  (* Index 09 of struct array *)
  ix10 : ULINT;  (* Index 10 of struct array *)
  ix11 : ULINT;  (* Index 11 of struct array *)
  ix12 : ULINT;  (* Index 12 of struct array *)
  ix13 : ULINT;  (* Index 13 of struct array *)
  ix14 : ULINT;  (* Index 14 of struct array *)
  ix15 : ULINT;  (* Index 15 of struct array *)
  ix16 : ULINT;  (* Index 16 of struct array *)
  ix17 : ULINT;  (* Index 17 of struct array *)
  ix18 : ULINT;  (* Index 18 of struct array *)
  ix19 : ULINT;  (* Index 19 of struct array *)
  ix20 : ULINT;  (* Index 20 of struct array *)
  ix21 : ULINT;  (* Index 21 of struct array *)
  ix22 : ULINT;  (* Index 22 of struct array *)
  ix23 : ULINT;  (* Index 23 of struct array *)
  ix24 : ULINT;  (* Index 24 of struct array *)
  ix25 : ULINT;  (* Index 25 of struct array *)
  ix26 : ULINT;  (* Index 26 of struct array *)
  ix27 : ULINT;  (* Index 27 of struct array *)
  ix28 : ULINT;  (* Index 28 of struct array *)
  ix29 : ULINT;  (* Index 29 of struct array *)
  ix30 : ULINT;  (* Index 30 of struct array *)
  ix31 : ULINT;  (* Index 31 of struct array *)
END_STRUCT;
END_TYPE

TYPE USINT32 : STRUCT
  ix00 : USINT;  (* Index 00 of struct array *)
  ix01 : USINT;  (* Index 01 of struct array *)
  ix02 : USINT;  (* Index 02 of struct array *)
  ix03 : USINT;  (* Index 03 of struct array *)
  ix04 : USINT;  (* Index 04 of struct array *)
  ix05 : USINT;  (* Index 05 of struct array *)
  ix06 : USINT;  (* Index 06 of struct array *)
  ix07 : USINT;  (* Index 07 of struct array *)
  ix08 : USINT;  (* Index 08 of struct array *)
  ix09 : USINT;  (* Index 09 of struct array *)
  ix10 : USINT;  (* Index 10 of struct array *)
  ix11 : USINT;  (* Index 11 of struct array *)
  ix12 : USINT;  (* Index 12 of struct array *)
  ix13 : USINT;  (* Index 13 of struct array *)
  ix14 : USINT;  (* Index 14 of struct array *)
  ix15 : USINT;  (* Index 15 of struct array *)
  ix16 : USINT;  (* Index 16 of struct array *)
  ix17 : USINT;  (* Index 17 of struct array *)
  ix18 : USINT;  (* Index 18 of struct array *)
  ix19 : USINT;  (* Index 19 of struct array *)
  ix20 : USINT;  (* Index 20 of struct array *)
  ix21 : USINT;  (* Index 21 of struct array *)
  ix22 : USINT;  (* Index 22 of struct array *)
  ix23 : USINT;  (* Index 23 of struct array *)
  ix24 : USINT;  (* Index 24 of struct array *)
  ix25 : USINT;  (* Index 25 of struct array *)
  ix26 : USINT;  (* Index 26 of struct array *)
  ix27 : USINT;  (* Index 27 of struct array *)
  ix28 : USINT;  (* Index 28 of struct array *)
  ix29 : USINT;  (* Index 29 of struct array *)
  ix30 : USINT;  (* Index 30 of struct array *)
  ix31 : USINT;  (* Index 31 of struct array *)
END_STRUCT;
END_TYPE

TYPE WORD32 : STRUCT
  ix00 : WORD;  (* Index 00 of struct array *)
  ix01 : WORD;  (* Index 01 of struct array *)
  ix02 : WORD;  (* Index 02 of struct array *)
  ix03 : WORD;  (* Index 03 of struct array *)
  ix04 : WORD;  (* Index 04 of struct array *)
  ix05 : WORD;  (* Index 05 of struct array *)
  ix06 : WORD;  (* Index 06 of struct array *)
  ix07 : WORD;  (* Index 07 of struct array *)
  ix08 : WORD;  (* Index 08 of struct array *)
  ix09 : WORD;  (* Index 09 of struct array *)
  ix10 : WORD;  (* Index 10 of struct array *)
  ix11 : WORD;  (* Index 11 of struct array *)
  ix12 : WORD;  (* Index 12 of struct array *)
  ix13 : WORD;  (* Index 13 of struct array *)
  ix14 : WORD;  (* Index 14 of struct array *)
  ix15 : WORD;  (* Index 15 of struct array *)
  ix16 : WORD;  (* Index 16 of struct array *)
  ix17 : WORD;  (* Index 17 of struct array *)
  ix18 : WORD;  (* Index 18 of struct array *)
  ix19 : WORD;  (* Index 19 of struct array *)
  ix20 : WORD;  (* Index 20 of struct array *)
  ix21 : WORD;  (* Index 21 of struct array *)
  ix22 : WORD;  (* Index 22 of struct array *)
  ix23 : WORD;  (* Index 23 of struct array *)
  ix24 : WORD;  (* Index 24 of struct array *)
  ix25 : WORD;  (* Index 25 of struct array *)
  ix26 : WORD;  (* Index 26 of struct array *)
  ix27 : WORD;  (* Index 27 of struct array *)
  ix28 : WORD;  (* Index 28 of struct array *)
  ix29 : WORD;  (* Index 29 of struct array *)
  ix30 : WORD;  (* Index 30 of struct array *)
  ix31 : WORD;  (* Index 31 of struct array *)
END_STRUCT;
END_TYPE

TYPE WSTRING32 : STRUCT
  ix00 : WSTRING;  (* Index 00 of struct array *)
  ix01 : WSTRING;  (* Index 01 of struct array *)
  ix02 : WSTRING;  (* Index 02 of struct array *)
  ix03 : WSTRING;  (* Index 03 of struct array *)
  ix04 : WSTRING;  (* Index 04 of struct array *)
  ix05 : WSTRING;  (* Index 05 of struct array *)
  ix06 : WSTRING;  (* Index 06 of struct array *)
  ix07 : WSTRING;  (* Index 07 of struct array *)
  ix08 : WSTRING;  (* Index 08 of struct array *)
  ix09 : WSTRING;  (* Index 09 of struct array *)
  ix10 : WSTRING;  (* Index 10 of struct array *)
  ix11 : WSTRING;  (* Index 11 of struct array *)
  ix12 : WSTRING;  (* Index 12 of struct array *)
  ix13 : WSTRING;  (* Index 13 of struct array *)
  ix14 : WSTRING;  (* Index 14 of struct array *)
  ix15 : WSTRING;  (* Index 15 of struct array *)
  ix16 : WSTRING;  (* Index 16 of struct array *)
  ix17 : WSTRING;  (* Index 17 of struct array *)
  ix18 : WSTRING;  (* Index 18 of struct array *)
  ix19 : WSTRING;  (* Index 19 of struct array *)
  ix20 : WSTRING;  (* Index 20 of struct array *)
  ix21 : WSTRING;  (* Index 21 of struct array *)
  ix22 : WSTRING;  (* Index 22 of struct array *)
  ix23 : WSTRING;  (* Index 23 of struct array *)
  ix24 : WSTRING;  (* Index 24 of struct array *)
  ix25 : WSTRING;  (* Index 25 of struct array *)
  ix26 : WSTRING;  (* Index 26 of struct array *)
  ix27 : WSTRING;  (* Index 27 of struct array *)
  ix28 : WSTRING;  (* Index 28 of struct array *)
  ix29 : WSTRING;  (* Index 29 of struct array *)
  ix30 : WSTRING;  (* Index 30 of struct array *)
  ix31 : WSTRING;  (* Index 31 of struct array *)
END_STRUCT;
END_TYPE

FUNCTION getBool32 : BOOL
  VAR_INPUT
    data : BOOL32;  (* Data to work on *)
    ix : USINT;  (* Index to retrieve *)
  END_VAR

            CASE ix OF
	0: getBool32 := data.ix00; (*Return index 0 for the data struct*)
	1: getBool32 := data.ix01; (*Return index 1 for the data struct*)
	2: getBool32 := data.ix02; (*Return index 2 for the data struct*)
	3: getBool32 := data.ix03; (*Return index 3 for the data struct*)
	4: getBool32 := data.ix04; (*Return index 4 for the data struct*)
	5: getBool32 := data.ix05; (*Return index 5 for the data struct*)
	6: getBool32 := data.ix06; (*Return index 6 for the data struct*)
	7: getBool32 := data.ix07; (*Return index 7 for the data struct*)
	8: getBool32 := data.ix08; (*Return index 8 for the data struct*)
	9: getBool32 := data.ix09; (*Return index 9 for the data struct*)
	10: getBool32 := data.ix10; (*Return index 10 for the data struct*)
	11: getBool32 := data.ix11; (*Return index 11 for the data struct*)
	12: getBool32 := data.ix12; (*Return index 12 for the data struct*)
	13: getBool32 := data.ix13; (*Return index 13 for the data struct*)
	14: getBool32 := data.ix14; (*Return index 14 for the data struct*)
	15: getBool32 := data.ix15; (*Return index 15 for the data struct*)
	16: getBool32 := data.ix16; (*Return index 16 for the data struct*)
	17: getBool32 := data.ix17; (*Return index 17 for the data struct*)
	18: getBool32 := data.ix18; (*Return index 18 for the data struct*)
	19: getBool32 := data.ix19; (*Return index 19 for the data struct*)
	20: getBool32 := data.ix20; (*Return index 20 for the data struct*)
	21: getBool32 := data.ix21; (*Return index 21 for the data struct*)
	22: getBool32 := data.ix22; (*Return index 22 for the data struct*)
	23: getBool32 := data.ix23; (*Return index 23 for the data struct*)
	24: getBool32 := data.ix24; (*Return index 24 for the data struct*)
	25: getBool32 := data.ix25; (*Return index 25 for the data struct*)
	26: getBool32 := data.ix26; (*Return index 26 for the data struct*)
	27: getBool32 := data.ix27; (*Return index 27 for the data struct*)
	28: getBool32 := data.ix28; (*Return index 28 for the data struct*)
	29: getBool32 := data.ix29; (*Return index 29 for the data struct*)
	30: getBool32 := data.ix30; (*Return index 30 for the data struct*)
	31: getBool32 := data.ix31; (*Return index 31 for the data struct*)
ELSE
	(*Index is invalid, return initial function value*)
	RETURN;
END_CASE
RETURN;

          
END_FUNCTION

FUNCTION getByte32 : BYTE
  VAR_INPUT
    data : BYTE32;  (* Data to work on *)
    ix : USINT;  (* Index to retrieve *)
  END_VAR

            CASE ix OF
	0: getByte32 := data.ix00; (*Return index 0 for the data struct*)
	1: getByte32 := data.ix01; (*Return index 1 for the data struct*)
	2: getByte32 := data.ix02; (*Return index 2 for the data struct*)
	3: getByte32 := data.ix03; (*Return index 3 for the data struct*)
	4: getByte32 := data.ix04; (*Return index 4 for the data struct*)
	5: getByte32 := data.ix05; (*Return index 5 for the data struct*)
	6: getByte32 := data.ix06; (*Return index 6 for the data struct*)
	7: getByte32 := data.ix07; (*Return index 7 for the data struct*)
	8: getByte32 := data.ix08; (*Return index 8 for the data struct*)
	9: getByte32 := data.ix09; (*Return index 9 for the data struct*)
	10: getByte32 := data.ix10; (*Return index 10 for the data struct*)
	11: getByte32 := data.ix11; (*Return index 11 for the data struct*)
	12: getByte32 := data.ix12; (*Return index 12 for the data struct*)
	13: getByte32 := data.ix13; (*Return index 13 for the data struct*)
	14: getByte32 := data.ix14; (*Return index 14 for the data struct*)
	15: getByte32 := data.ix15; (*Return index 15 for the data struct*)
	16: getByte32 := data.ix16; (*Return index 16 for the data struct*)
	17: getByte32 := data.ix17; (*Return index 17 for the data struct*)
	18: getByte32 := data.ix18; (*Return index 18 for the data struct*)
	19: getByte32 := data.ix19; (*Return index 19 for the data struct*)
	20: getByte32 := data.ix20; (*Return index 20 for the data struct*)
	21: getByte32 := data.ix21; (*Return index 21 for the data struct*)
	22: getByte32 := data.ix22; (*Return index 22 for the data struct*)
	23: getByte32 := data.ix23; (*Return index 23 for the data struct*)
	24: getByte32 := data.ix24; (*Return index 24 for the data struct*)
	25: getByte32 := data.ix25; (*Return index 25 for the data struct*)
	26: getByte32 := data.ix26; (*Return index 26 for the data struct*)
	27: getByte32 := data.ix27; (*Return index 27 for the data struct*)
	28: getByte32 := data.ix28; (*Return index 28 for the data struct*)
	29: getByte32 := data.ix29; (*Return index 29 for the data struct*)
	30: getByte32 := data.ix30; (*Return index 30 for the data struct*)
	31: getByte32 := data.ix31; (*Return index 31 for the data struct*)
ELSE
	(*Index is invalid, return initial function value*)
	RETURN;
END_CASE
RETURN;

          
END_FUNCTION

FUNCTION getDate_and_time32 : DT
  VAR_INPUT
    data : DATE_AND_TIME32;  (* Data to work on *)
    ix : USINT;  (* Index to retrieve *)
  END_VAR

            CASE ix OF
	0: getDate_and_time32 := data.ix00; (*Return index 0 for the data struct*)
	1: getDate_and_time32 := data.ix01; (*Return index 1 for the data struct*)
	2: getDate_and_time32 := data.ix02; (*Return index 2 for the data struct*)
	3: getDate_and_time32 := data.ix03; (*Return index 3 for the data struct*)
	4: getDate_and_time32 := data.ix04; (*Return index 4 for the data struct*)
	5: getDate_and_time32 := data.ix05; (*Return index 5 for the data struct*)
	6: getDate_and_time32 := data.ix06; (*Return index 6 for the data struct*)
	7: getDate_and_time32 := data.ix07; (*Return index 7 for the data struct*)
	8: getDate_and_time32 := data.ix08; (*Return index 8 for the data struct*)
	9: getDate_and_time32 := data.ix09; (*Return index 9 for the data struct*)
	10: getDate_and_time32 := data.ix10; (*Return index 10 for the data struct*)
	11: getDate_and_time32 := data.ix11; (*Return index 11 for the data struct*)
	12: getDate_and_time32 := data.ix12; (*Return index 12 for the data struct*)
	13: getDate_and_time32 := data.ix13; (*Return index 13 for the data struct*)
	14: getDate_and_time32 := data.ix14; (*Return index 14 for the data struct*)
	15: getDate_and_time32 := data.ix15; (*Return index 15 for the data struct*)
	16: getDate_and_time32 := data.ix16; (*Return index 16 for the data struct*)
	17: getDate_and_time32 := data.ix17; (*Return index 17 for the data struct*)
	18: getDate_and_time32 := data.ix18; (*Return index 18 for the data struct*)
	19: getDate_and_time32 := data.ix19; (*Return index 19 for the data struct*)
	20: getDate_and_time32 := data.ix20; (*Return index 20 for the data struct*)
	21: getDate_and_time32 := data.ix21; (*Return index 21 for the data struct*)
	22: getDate_and_time32 := data.ix22; (*Return index 22 for the data struct*)
	23: getDate_and_time32 := data.ix23; (*Return index 23 for the data struct*)
	24: getDate_and_time32 := data.ix24; (*Return index 24 for the data struct*)
	25: getDate_and_time32 := data.ix25; (*Return index 25 for the data struct*)
	26: getDate_and_time32 := data.ix26; (*Return index 26 for the data struct*)
	27: getDate_and_time32 := data.ix27; (*Return index 27 for the data struct*)
	28: getDate_and_time32 := data.ix28; (*Return index 28 for the data struct*)
	29: getDate_and_time32 := data.ix29; (*Return index 29 for the data struct*)
	30: getDate_and_time32 := data.ix30; (*Return index 30 for the data struct*)
	31: getDate_and_time32 := data.ix31; (*Return index 31 for the data struct*)
ELSE
	(*Index is invalid, return initial function value*)
	RETURN;
END_CASE
RETURN;

          
END_FUNCTION

FUNCTION getDate32 : DATE
  VAR_INPUT
    data : DATE32;  (* Data to work on *)
    ix : USINT;  (* Index to retrieve *)
  END_VAR

            CASE ix OF
	0: getDate32 := data.ix00; (*Return index 0 for the data struct*)
	1: getDate32 := data.ix01; (*Return index 1 for the data struct*)
	2: getDate32 := data.ix02; (*Return index 2 for the data struct*)
	3: getDate32 := data.ix03; (*Return index 3 for the data struct*)
	4: getDate32 := data.ix04; (*Return index 4 for the data struct*)
	5: getDate32 := data.ix05; (*Return index 5 for the data struct*)
	6: getDate32 := data.ix06; (*Return index 6 for the data struct*)
	7: getDate32 := data.ix07; (*Return index 7 for the data struct*)
	8: getDate32 := data.ix08; (*Return index 8 for the data struct*)
	9: getDate32 := data.ix09; (*Return index 9 for the data struct*)
	10: getDate32 := data.ix10; (*Return index 10 for the data struct*)
	11: getDate32 := data.ix11; (*Return index 11 for the data struct*)
	12: getDate32 := data.ix12; (*Return index 12 for the data struct*)
	13: getDate32 := data.ix13; (*Return index 13 for the data struct*)
	14: getDate32 := data.ix14; (*Return index 14 for the data struct*)
	15: getDate32 := data.ix15; (*Return index 15 for the data struct*)
	16: getDate32 := data.ix16; (*Return index 16 for the data struct*)
	17: getDate32 := data.ix17; (*Return index 17 for the data struct*)
	18: getDate32 := data.ix18; (*Return index 18 for the data struct*)
	19: getDate32 := data.ix19; (*Return index 19 for the data struct*)
	20: getDate32 := data.ix20; (*Return index 20 for the data struct*)
	21: getDate32 := data.ix21; (*Return index 21 for the data struct*)
	22: getDate32 := data.ix22; (*Return index 22 for the data struct*)
	23: getDate32 := data.ix23; (*Return index 23 for the data struct*)
	24: getDate32 := data.ix24; (*Return index 24 for the data struct*)
	25: getDate32 := data.ix25; (*Return index 25 for the data struct*)
	26: getDate32 := data.ix26; (*Return index 26 for the data struct*)
	27: getDate32 := data.ix27; (*Return index 27 for the data struct*)
	28: getDate32 := data.ix28; (*Return index 28 for the data struct*)
	29: getDate32 := data.ix29; (*Return index 29 for the data struct*)
	30: getDate32 := data.ix30; (*Return index 30 for the data struct*)
	31: getDate32 := data.ix31; (*Return index 31 for the data struct*)
ELSE
	(*Index is invalid, return initial function value*)
	RETURN;
END_CASE
RETURN;
          
END_FUNCTION

FUNCTION getDint32 : DINT
  VAR_INPUT
    data : DINT32;  (* Data to work on *)
    ix : USINT;  (* Index to retrieve *)
  END_VAR

            CASE ix OF
	0: getDint32 := data.ix00; (*Return index 0 for the data struct*)
	1: getDint32 := data.ix01; (*Return index 1 for the data struct*)
	2: getDint32 := data.ix02; (*Return index 2 for the data struct*)
	3: getDint32 := data.ix03; (*Return index 3 for the data struct*)
	4: getDint32 := data.ix04; (*Return index 4 for the data struct*)
	5: getDint32 := data.ix05; (*Return index 5 for the data struct*)
	6: getDint32 := data.ix06; (*Return index 6 for the data struct*)
	7: getDint32 := data.ix07; (*Return index 7 for the data struct*)
	8: getDint32 := data.ix08; (*Return index 8 for the data struct*)
	9: getDint32 := data.ix09; (*Return index 9 for the data struct*)
	10: getDint32 := data.ix10; (*Return index 10 for the data struct*)
	11: getDint32 := data.ix11; (*Return index 11 for the data struct*)
	12: getDint32 := data.ix12; (*Return index 12 for the data struct*)
	13: getDint32 := data.ix13; (*Return index 13 for the data struct*)
	14: getDint32 := data.ix14; (*Return index 14 for the data struct*)
	15: getDint32 := data.ix15; (*Return index 15 for the data struct*)
	16: getDint32 := data.ix16; (*Return index 16 for the data struct*)
	17: getDint32 := data.ix17; (*Return index 17 for the data struct*)
	18: getDint32 := data.ix18; (*Return index 18 for the data struct*)
	19: getDint32 := data.ix19; (*Return index 19 for the data struct*)
	20: getDint32 := data.ix20; (*Return index 20 for the data struct*)
	21: getDint32 := data.ix21; (*Return index 21 for the data struct*)
	22: getDint32 := data.ix22; (*Return index 22 for the data struct*)
	23: getDint32 := data.ix23; (*Return index 23 for the data struct*)
	24: getDint32 := data.ix24; (*Return index 24 for the data struct*)
	25: getDint32 := data.ix25; (*Return index 25 for the data struct*)
	26: getDint32 := data.ix26; (*Return index 26 for the data struct*)
	27: getDint32 := data.ix27; (*Return index 27 for the data struct*)
	28: getDint32 := data.ix28; (*Return index 28 for the data struct*)
	29: getDint32 := data.ix29; (*Return index 29 for the data struct*)
	30: getDint32 := data.ix30; (*Return index 30 for the data struct*)
	31: getDint32 := data.ix31; (*Return index 31 for the data struct*)
ELSE
	(*Index is invalid, return initial function value*)
	RETURN;
END_CASE
RETURN;

          
END_FUNCTION

FUNCTION getDword32 : DWORD
  VAR_INPUT
    data : DWORD32;  (* Data to work on *)
    ix : USINT;  (* Index to retrieve *)
  END_VAR

            CASE ix OF
	0: getDword32 := data.ix00; (*Return index 0 for the data struct*)
	1: getDword32 := data.ix01; (*Return index 1 for the data struct*)
	2: getDword32 := data.ix02; (*Return index 2 for the data struct*)
	3: getDword32 := data.ix03; (*Return index 3 for the data struct*)
	4: getDword32 := data.ix04; (*Return index 4 for the data struct*)
	5: getDword32 := data.ix05; (*Return index 5 for the data struct*)
	6: getDword32 := data.ix06; (*Return index 6 for the data struct*)
	7: getDword32 := data.ix07; (*Return index 7 for the data struct*)
	8: getDword32 := data.ix08; (*Return index 8 for the data struct*)
	9: getDword32 := data.ix09; (*Return index 9 for the data struct*)
	10: getDword32 := data.ix10; (*Return index 10 for the data struct*)
	11: getDword32 := data.ix11; (*Return index 11 for the data struct*)
	12: getDword32 := data.ix12; (*Return index 12 for the data struct*)
	13: getDword32 := data.ix13; (*Return index 13 for the data struct*)
	14: getDword32 := data.ix14; (*Return index 14 for the data struct*)
	15: getDword32 := data.ix15; (*Return index 15 for the data struct*)
	16: getDword32 := data.ix16; (*Return index 16 for the data struct*)
	17: getDword32 := data.ix17; (*Return index 17 for the data struct*)
	18: getDword32 := data.ix18; (*Return index 18 for the data struct*)
	19: getDword32 := data.ix19; (*Return index 19 for the data struct*)
	20: getDword32 := data.ix20; (*Return index 20 for the data struct*)
	21: getDword32 := data.ix21; (*Return index 21 for the data struct*)
	22: getDword32 := data.ix22; (*Return index 22 for the data struct*)
	23: getDword32 := data.ix23; (*Return index 23 for the data struct*)
	24: getDword32 := data.ix24; (*Return index 24 for the data struct*)
	25: getDword32 := data.ix25; (*Return index 25 for the data struct*)
	26: getDword32 := data.ix26; (*Return index 26 for the data struct*)
	27: getDword32 := data.ix27; (*Return index 27 for the data struct*)
	28: getDword32 := data.ix28; (*Return index 28 for the data struct*)
	29: getDword32 := data.ix29; (*Return index 29 for the data struct*)
	30: getDword32 := data.ix30; (*Return index 30 for the data struct*)
	31: getDword32 := data.ix31; (*Return index 31 for the data struct*)
ELSE
	(*Index is invalid, return initial function value*)
	RETURN;
END_CASE
RETURN;

          
END_FUNCTION

FUNCTION getInt32 : INT
  VAR_INPUT
    data : INT32;  (* Data to work on *)
    ix : USINT;  (* Index to retrieve *)
  END_VAR

            CASE ix OF
	0: getInt32 := data.ix00; (*Return index 0 for the data struct*)
	1: getInt32 := data.ix01; (*Return index 1 for the data struct*)
	2: getInt32 := data.ix02; (*Return index 2 for the data struct*)
	3: getInt32 := data.ix03; (*Return index 3 for the data struct*)
	4: getInt32 := data.ix04; (*Return index 4 for the data struct*)
	5: getInt32 := data.ix05; (*Return index 5 for the data struct*)
	6: getInt32 := data.ix06; (*Return index 6 for the data struct*)
	7: getInt32 := data.ix07; (*Return index 7 for the data struct*)
	8: getInt32 := data.ix08; (*Return index 8 for the data struct*)
	9: getInt32 := data.ix09; (*Return index 9 for the data struct*)
	10: getInt32 := data.ix10; (*Return index 10 for the data struct*)
	11: getInt32 := data.ix11; (*Return index 11 for the data struct*)
	12: getInt32 := data.ix12; (*Return index 12 for the data struct*)
	13: getInt32 := data.ix13; (*Return index 13 for the data struct*)
	14: getInt32 := data.ix14; (*Return index 14 for the data struct*)
	15: getInt32 := data.ix15; (*Return index 15 for the data struct*)
	16: getInt32 := data.ix16; (*Return index 16 for the data struct*)
	17: getInt32 := data.ix17; (*Return index 17 for the data struct*)
	18: getInt32 := data.ix18; (*Return index 18 for the data struct*)
	19: getInt32 := data.ix19; (*Return index 19 for the data struct*)
	20: getInt32 := data.ix20; (*Return index 20 for the data struct*)
	21: getInt32 := data.ix21; (*Return index 21 for the data struct*)
	22: getInt32 := data.ix22; (*Return index 22 for the data struct*)
	23: getInt32 := data.ix23; (*Return index 23 for the data struct*)
	24: getInt32 := data.ix24; (*Return index 24 for the data struct*)
	25: getInt32 := data.ix25; (*Return index 25 for the data struct*)
	26: getInt32 := data.ix26; (*Return index 26 for the data struct*)
	27: getInt32 := data.ix27; (*Return index 27 for the data struct*)
	28: getInt32 := data.ix28; (*Return index 28 for the data struct*)
	29: getInt32 := data.ix29; (*Return index 29 for the data struct*)
	30: getInt32 := data.ix30; (*Return index 30 for the data struct*)
	31: getInt32 := data.ix31; (*Return index 31 for the data struct*)
ELSE
	(*Index is invalid, return initial function value*)
	RETURN;
END_CASE
RETURN;

          
END_FUNCTION

FUNCTION getLdate_and_time32 : LDATE_AND_TIME
  VAR_INPUT
    data : LDATE_AND_TIME32;  (* Data to work on *)
    ix : USINT;  (* Index to retrieve *)
  END_VAR

            CASE ix OF
	0: getLdate_and_time32 := data.ix00; (*Return index 0 for the data struct*)
	1: getLdate_and_time32 := data.ix01; (*Return index 1 for the data struct*)
	2: getLdate_and_time32 := data.ix02; (*Return index 2 for the data struct*)
	3: getLdate_and_time32 := data.ix03; (*Return index 3 for the data struct*)
	4: getLdate_and_time32 := data.ix04; (*Return index 4 for the data struct*)
	5: getLdate_and_time32 := data.ix05; (*Return index 5 for the data struct*)
	6: getLdate_and_time32 := data.ix06; (*Return index 6 for the data struct*)
	7: getLdate_and_time32 := data.ix07; (*Return index 7 for the data struct*)
	8: getLdate_and_time32 := data.ix08; (*Return index 8 for the data struct*)
	9: getLdate_and_time32 := data.ix09; (*Return index 9 for the data struct*)
	10: getLdate_and_time32 := data.ix10; (*Return index 10 for the data struct*)
	11: getLdate_and_time32 := data.ix11; (*Return index 11 for the data struct*)
	12: getLdate_and_time32 := data.ix12; (*Return index 12 for the data struct*)
	13: getLdate_and_time32 := data.ix13; (*Return index 13 for the data struct*)
	14: getLdate_and_time32 := data.ix14; (*Return index 14 for the data struct*)
	15: getLdate_and_time32 := data.ix15; (*Return index 15 for the data struct*)
	16: getLdate_and_time32 := data.ix16; (*Return index 16 for the data struct*)
	17: getLdate_and_time32 := data.ix17; (*Return index 17 for the data struct*)
	18: getLdate_and_time32 := data.ix18; (*Return index 18 for the data struct*)
	19: getLdate_and_time32 := data.ix19; (*Return index 19 for the data struct*)
	20: getLdate_and_time32 := data.ix20; (*Return index 20 for the data struct*)
	21: getLdate_and_time32 := data.ix21; (*Return index 21 for the data struct*)
	22: getLdate_and_time32 := data.ix22; (*Return index 22 for the data struct*)
	23: getLdate_and_time32 := data.ix23; (*Return index 23 for the data struct*)
	24: getLdate_and_time32 := data.ix24; (*Return index 24 for the data struct*)
	25: getLdate_and_time32 := data.ix25; (*Return index 25 for the data struct*)
	26: getLdate_and_time32 := data.ix26; (*Return index 26 for the data struct*)
	27: getLdate_and_time32 := data.ix27; (*Return index 27 for the data struct*)
	28: getLdate_and_time32 := data.ix28; (*Return index 28 for the data struct*)
	29: getLdate_and_time32 := data.ix29; (*Return index 29 for the data struct*)
	30: getLdate_and_time32 := data.ix30; (*Return index 30 for the data struct*)
	31: getLdate_and_time32 := data.ix31; (*Return index 31 for the data struct*)
ELSE
	(*Index is invalid, return initial function value*)
	RETURN;
END_CASE
RETURN;

          
END_FUNCTION

FUNCTION getLdate32 : LDATE
  VAR_INPUT
    data : LDATE32;  (* Data to work on *)
    ix : USINT;  (* Index to retrieve *)
  END_VAR

            CASE ix OF
	0: getLdate32 := data.ix00; (*Return index 0 for the data struct*)
	1: getLdate32 := data.ix01; (*Return index 1 for the data struct*)
	2: getLdate32 := data.ix02; (*Return index 2 for the data struct*)
	3: getLdate32 := data.ix03; (*Return index 3 for the data struct*)
	4: getLdate32 := data.ix04; (*Return index 4 for the data struct*)
	5: getLdate32 := data.ix05; (*Return index 5 for the data struct*)
	6: getLdate32 := data.ix06; (*Return index 6 for the data struct*)
	7: getLdate32 := data.ix07; (*Return index 7 for the data struct*)
	8: getLdate32 := data.ix08; (*Return index 8 for the data struct*)
	9: getLdate32 := data.ix09; (*Return index 9 for the data struct*)
	10: getLdate32 := data.ix10; (*Return index 10 for the data struct*)
	11: getLdate32 := data.ix11; (*Return index 11 for the data struct*)
	12: getLdate32 := data.ix12; (*Return index 12 for the data struct*)
	13: getLdate32 := data.ix13; (*Return index 13 for the data struct*)
	14: getLdate32 := data.ix14; (*Return index 14 for the data struct*)
	15: getLdate32 := data.ix15; (*Return index 15 for the data struct*)
	16: getLdate32 := data.ix16; (*Return index 16 for the data struct*)
	17: getLdate32 := data.ix17; (*Return index 17 for the data struct*)
	18: getLdate32 := data.ix18; (*Return index 18 for the data struct*)
	19: getLdate32 := data.ix19; (*Return index 19 for the data struct*)
	20: getLdate32 := data.ix20; (*Return index 20 for the data struct*)
	21: getLdate32 := data.ix21; (*Return index 21 for the data struct*)
	22: getLdate32 := data.ix22; (*Return index 22 for the data struct*)
	23: getLdate32 := data.ix23; (*Return index 23 for the data struct*)
	24: getLdate32 := data.ix24; (*Return index 24 for the data struct*)
	25: getLdate32 := data.ix25; (*Return index 25 for the data struct*)
	26: getLdate32 := data.ix26; (*Return index 26 for the data struct*)
	27: getLdate32 := data.ix27; (*Return index 27 for the data struct*)
	28: getLdate32 := data.ix28; (*Return index 28 for the data struct*)
	29: getLdate32 := data.ix29; (*Return index 29 for the data struct*)
	30: getLdate32 := data.ix30; (*Return index 30 for the data struct*)
	31: getLdate32 := data.ix31; (*Return index 31 for the data struct*)
ELSE
	(*Index is invalid, return initial function value*)
	RETURN;
END_CASE
RETURN;

          
END_FUNCTION

FUNCTION getLint32 : LINT
  VAR_INPUT
    data : LINT32;  (* Data to work on *)
    ix : USINT;  (* Index to retrieve *)
  END_VAR

            CASE ix OF
	0: getLint32 := data.ix00; (*Return index 0 for the data struct*)
	1: getLint32 := data.ix01; (*Return index 1 for the data struct*)
	2: getLint32 := data.ix02; (*Return index 2 for the data struct*)
	3: getLint32 := data.ix03; (*Return index 3 for the data struct*)
	4: getLint32 := data.ix04; (*Return index 4 for the data struct*)
	5: getLint32 := data.ix05; (*Return index 5 for the data struct*)
	6: getLint32 := data.ix06; (*Return index 6 for the data struct*)
	7: getLint32 := data.ix07; (*Return index 7 for the data struct*)
	8: getLint32 := data.ix08; (*Return index 8 for the data struct*)
	9: getLint32 := data.ix09; (*Return index 9 for the data struct*)
	10: getLint32 := data.ix10; (*Return index 10 for the data struct*)
	11: getLint32 := data.ix11; (*Return index 11 for the data struct*)
	12: getLint32 := data.ix12; (*Return index 12 for the data struct*)
	13: getLint32 := data.ix13; (*Return index 13 for the data struct*)
	14: getLint32 := data.ix14; (*Return index 14 for the data struct*)
	15: getLint32 := data.ix15; (*Return index 15 for the data struct*)
	16: getLint32 := data.ix16; (*Return index 16 for the data struct*)
	17: getLint32 := data.ix17; (*Return index 17 for the data struct*)
	18: getLint32 := data.ix18; (*Return index 18 for the data struct*)
	19: getLint32 := data.ix19; (*Return index 19 for the data struct*)
	20: getLint32 := data.ix20; (*Return index 20 for the data struct*)
	21: getLint32 := data.ix21; (*Return index 21 for the data struct*)
	22: getLint32 := data.ix22; (*Return index 22 for the data struct*)
	23: getLint32 := data.ix23; (*Return index 23 for the data struct*)
	24: getLint32 := data.ix24; (*Return index 24 for the data struct*)
	25: getLint32 := data.ix25; (*Return index 25 for the data struct*)
	26: getLint32 := data.ix26; (*Return index 26 for the data struct*)
	27: getLint32 := data.ix27; (*Return index 27 for the data struct*)
	28: getLint32 := data.ix28; (*Return index 28 for the data struct*)
	29: getLint32 := data.ix29; (*Return index 29 for the data struct*)
	30: getLint32 := data.ix30; (*Return index 30 for the data struct*)
	31: getLint32 := data.ix31; (*Return index 31 for the data struct*)
ELSE
	(*Index is invalid, return initial function value*)
	RETURN;
END_CASE
RETURN;

          
END_FUNCTION

FUNCTION getLreal32 : LREAL
  VAR_INPUT
    data : LREAL32;  (* Data to work on *)
    ix : USINT;  (* Index to retrieve *)
  END_VAR

            CASE ix OF
	0: getLreal32 := data.ix00; (*Return index 0 for the data struct*)
	1: getLreal32 := data.ix01; (*Return index 1 for the data struct*)
	2: getLreal32 := data.ix02; (*Return index 2 for the data struct*)
	3: getLreal32 := data.ix03; (*Return index 3 for the data struct*)
	4: getLreal32 := data.ix04; (*Return index 4 for the data struct*)
	5: getLreal32 := data.ix05; (*Return index 5 for the data struct*)
	6: getLreal32 := data.ix06; (*Return index 6 for the data struct*)
	7: getLreal32 := data.ix07; (*Return index 7 for the data struct*)
	8: getLreal32 := data.ix08; (*Return index 8 for the data struct*)
	9: getLreal32 := data.ix09; (*Return index 9 for the data struct*)
	10: getLreal32 := data.ix10; (*Return index 10 for the data struct*)
	11: getLreal32 := data.ix11; (*Return index 11 for the data struct*)
	12: getLreal32 := data.ix12; (*Return index 12 for the data struct*)
	13: getLreal32 := data.ix13; (*Return index 13 for the data struct*)
	14: getLreal32 := data.ix14; (*Return index 14 for the data struct*)
	15: getLreal32 := data.ix15; (*Return index 15 for the data struct*)
	16: getLreal32 := data.ix16; (*Return index 16 for the data struct*)
	17: getLreal32 := data.ix17; (*Return index 17 for the data struct*)
	18: getLreal32 := data.ix18; (*Return index 18 for the data struct*)
	19: getLreal32 := data.ix19; (*Return index 19 for the data struct*)
	20: getLreal32 := data.ix20; (*Return index 20 for the data struct*)
	21: getLreal32 := data.ix21; (*Return index 21 for the data struct*)
	22: getLreal32 := data.ix22; (*Return index 22 for the data struct*)
	23: getLreal32 := data.ix23; (*Return index 23 for the data struct*)
	24: getLreal32 := data.ix24; (*Return index 24 for the data struct*)
	25: getLreal32 := data.ix25; (*Return index 25 for the data struct*)
	26: getLreal32 := data.ix26; (*Return index 26 for the data struct*)
	27: getLreal32 := data.ix27; (*Return index 27 for the data struct*)
	28: getLreal32 := data.ix28; (*Return index 28 for the data struct*)
	29: getLreal32 := data.ix29; (*Return index 29 for the data struct*)
	30: getLreal32 := data.ix30; (*Return index 30 for the data struct*)
	31: getLreal32 := data.ix31; (*Return index 31 for the data struct*)
ELSE
	(*Index is invalid, return initial function value*)
	RETURN;
END_CASE
RETURN;

          
END_FUNCTION

FUNCTION getLtime_of_day32 : LTIME_OF_DAY
  VAR_INPUT
    data : LTIME_OF_DAY32;  (* Data to work on *)
    ix : USINT;  (* Index to retrieve *)
  END_VAR

            CASE ix OF
	0: getLtime_of_day32 := data.ix00; (*Return index 0 for the data struct*)
	1: getLtime_of_day32 := data.ix01; (*Return index 1 for the data struct*)
	2: getLtime_of_day32 := data.ix02; (*Return index 2 for the data struct*)
	3: getLtime_of_day32 := data.ix03; (*Return index 3 for the data struct*)
	4: getLtime_of_day32 := data.ix04; (*Return index 4 for the data struct*)
	5: getLtime_of_day32 := data.ix05; (*Return index 5 for the data struct*)
	6: getLtime_of_day32 := data.ix06; (*Return index 6 for the data struct*)
	7: getLtime_of_day32 := data.ix07; (*Return index 7 for the data struct*)
	8: getLtime_of_day32 := data.ix08; (*Return index 8 for the data struct*)
	9: getLtime_of_day32 := data.ix09; (*Return index 9 for the data struct*)
	10: getLtime_of_day32 := data.ix10; (*Return index 10 for the data struct*)
	11: getLtime_of_day32 := data.ix11; (*Return index 11 for the data struct*)
	12: getLtime_of_day32 := data.ix12; (*Return index 12 for the data struct*)
	13: getLtime_of_day32 := data.ix13; (*Return index 13 for the data struct*)
	14: getLtime_of_day32 := data.ix14; (*Return index 14 for the data struct*)
	15: getLtime_of_day32 := data.ix15; (*Return index 15 for the data struct*)
	16: getLtime_of_day32 := data.ix16; (*Return index 16 for the data struct*)
	17: getLtime_of_day32 := data.ix17; (*Return index 17 for the data struct*)
	18: getLtime_of_day32 := data.ix18; (*Return index 18 for the data struct*)
	19: getLtime_of_day32 := data.ix19; (*Return index 19 for the data struct*)
	20: getLtime_of_day32 := data.ix20; (*Return index 20 for the data struct*)
	21: getLtime_of_day32 := data.ix21; (*Return index 21 for the data struct*)
	22: getLtime_of_day32 := data.ix22; (*Return index 22 for the data struct*)
	23: getLtime_of_day32 := data.ix23; (*Return index 23 for the data struct*)
	24: getLtime_of_day32 := data.ix24; (*Return index 24 for the data struct*)
	25: getLtime_of_day32 := data.ix25; (*Return index 25 for the data struct*)
	26: getLtime_of_day32 := data.ix26; (*Return index 26 for the data struct*)
	27: getLtime_of_day32 := data.ix27; (*Return index 27 for the data struct*)
	28: getLtime_of_day32 := data.ix28; (*Return index 28 for the data struct*)
	29: getLtime_of_day32 := data.ix29; (*Return index 29 for the data struct*)
	30: getLtime_of_day32 := data.ix30; (*Return index 30 for the data struct*)
	31: getLtime_of_day32 := data.ix31; (*Return index 31 for the data struct*)
ELSE
	(*Index is invalid, return initial function value*)
	RETURN;
END_CASE
RETURN;

          
END_FUNCTION

FUNCTION getLtime32 : LTIME
  VAR_INPUT
    data : LTIME32;  (* Data to work on *)
    ix : USINT;  (* Index to retrieve *)
  END_VAR

            CASE ix OF
	0: getLtime32 := data.ix00; (*Return index 0 for the data struct*)
	1: getLtime32 := data.ix01; (*Return index 1 for the data struct*)
	2: getLtime32 := data.ix02; (*Return index 2 for the data struct*)
	3: getLtime32 := data.ix03; (*Return index 3 for the data struct*)
	4: getLtime32 := data.ix04; (*Return index 4 for the data struct*)
	5: getLtime32 := data.ix05; (*Return index 5 for the data struct*)
	6: getLtime32 := data.ix06; (*Return index 6 for the data struct*)
	7: getLtime32 := data.ix07; (*Return index 7 for the data struct*)
	8: getLtime32 := data.ix08; (*Return index 8 for the data struct*)
	9: getLtime32 := data.ix09; (*Return index 9 for the data struct*)
	10: getLtime32 := data.ix10; (*Return index 10 for the data struct*)
	11: getLtime32 := data.ix11; (*Return index 11 for the data struct*)
	12: getLtime32 := data.ix12; (*Return index 12 for the data struct*)
	13: getLtime32 := data.ix13; (*Return index 13 for the data struct*)
	14: getLtime32 := data.ix14; (*Return index 14 for the data struct*)
	15: getLtime32 := data.ix15; (*Return index 15 for the data struct*)
	16: getLtime32 := data.ix16; (*Return index 16 for the data struct*)
	17: getLtime32 := data.ix17; (*Return index 17 for the data struct*)
	18: getLtime32 := data.ix18; (*Return index 18 for the data struct*)
	19: getLtime32 := data.ix19; (*Return index 19 for the data struct*)
	20: getLtime32 := data.ix20; (*Return index 20 for the data struct*)
	21: getLtime32 := data.ix21; (*Return index 21 for the data struct*)
	22: getLtime32 := data.ix22; (*Return index 22 for the data struct*)
	23: getLtime32 := data.ix23; (*Return index 23 for the data struct*)
	24: getLtime32 := data.ix24; (*Return index 24 for the data struct*)
	25: getLtime32 := data.ix25; (*Return index 25 for the data struct*)
	26: getLtime32 := data.ix26; (*Return index 26 for the data struct*)
	27: getLtime32 := data.ix27; (*Return index 27 for the data struct*)
	28: getLtime32 := data.ix28; (*Return index 28 for the data struct*)
	29: getLtime32 := data.ix29; (*Return index 29 for the data struct*)
	30: getLtime32 := data.ix30; (*Return index 30 for the data struct*)
	31: getLtime32 := data.ix31; (*Return index 31 for the data struct*)
ELSE
	(*Index is invalid, return initial function value*)
	RETURN;
END_CASE
RETURN;

          
END_FUNCTION

FUNCTION getLword32 : LWORD
  VAR_INPUT
    data : LWORD32;  (* Data to work on *)
    ix : USINT;  (* Index to retrieve *)
  END_VAR

            CASE ix OF
	0: getLword32 := data.ix00; (*Return index 0 for the data struct*)
	1: getLword32 := data.ix01; (*Return index 1 for the data struct*)
	2: getLword32 := data.ix02; (*Return index 2 for the data struct*)
	3: getLword32 := data.ix03; (*Return index 3 for the data struct*)
	4: getLword32 := data.ix04; (*Return index 4 for the data struct*)
	5: getLword32 := data.ix05; (*Return index 5 for the data struct*)
	6: getLword32 := data.ix06; (*Return index 6 for the data struct*)
	7: getLword32 := data.ix07; (*Return index 7 for the data struct*)
	8: getLword32 := data.ix08; (*Return index 8 for the data struct*)
	9: getLword32 := data.ix09; (*Return index 9 for the data struct*)
	10: getLword32 := data.ix10; (*Return index 10 for the data struct*)
	11: getLword32 := data.ix11; (*Return index 11 for the data struct*)
	12: getLword32 := data.ix12; (*Return index 12 for the data struct*)
	13: getLword32 := data.ix13; (*Return index 13 for the data struct*)
	14: getLword32 := data.ix14; (*Return index 14 for the data struct*)
	15: getLword32 := data.ix15; (*Return index 15 for the data struct*)
	16: getLword32 := data.ix16; (*Return index 16 for the data struct*)
	17: getLword32 := data.ix17; (*Return index 17 for the data struct*)
	18: getLword32 := data.ix18; (*Return index 18 for the data struct*)
	19: getLword32 := data.ix19; (*Return index 19 for the data struct*)
	20: getLword32 := data.ix20; (*Return index 20 for the data struct*)
	21: getLword32 := data.ix21; (*Return index 21 for the data struct*)
	22: getLword32 := data.ix22; (*Return index 22 for the data struct*)
	23: getLword32 := data.ix23; (*Return index 23 for the data struct*)
	24: getLword32 := data.ix24; (*Return index 24 for the data struct*)
	25: getLword32 := data.ix25; (*Return index 25 for the data struct*)
	26: getLword32 := data.ix26; (*Return index 26 for the data struct*)
	27: getLword32 := data.ix27; (*Return index 27 for the data struct*)
	28: getLword32 := data.ix28; (*Return index 28 for the data struct*)
	29: getLword32 := data.ix29; (*Return index 29 for the data struct*)
	30: getLword32 := data.ix30; (*Return index 30 for the data struct*)
	31: getLword32 := data.ix31; (*Return index 31 for the data struct*)
ELSE
	(*Index is invalid, return initial function value*)
	RETURN;
END_CASE
RETURN;

          
END_FUNCTION

FUNCTION getReal32 : REAL
  VAR_INPUT
    data : REAL32;  (* Data to work on *)
    ix : USINT;  (* Index to retrieve *)
  END_VAR

            CASE ix OF
	0: getReal32 := data.ix00; (*Return index 0 for the data struct*)
	1: getReal32 := data.ix01; (*Return index 1 for the data struct*)
	2: getReal32 := data.ix02; (*Return index 2 for the data struct*)
	3: getReal32 := data.ix03; (*Return index 3 for the data struct*)
	4: getReal32 := data.ix04; (*Return index 4 for the data struct*)
	5: getReal32 := data.ix05; (*Return index 5 for the data struct*)
	6: getReal32 := data.ix06; (*Return index 6 for the data struct*)
	7: getReal32 := data.ix07; (*Return index 7 for the data struct*)
	8: getReal32 := data.ix08; (*Return index 8 for the data struct*)
	9: getReal32 := data.ix09; (*Return index 9 for the data struct*)
	10: getReal32 := data.ix10; (*Return index 10 for the data struct*)
	11: getReal32 := data.ix11; (*Return index 11 for the data struct*)
	12: getReal32 := data.ix12; (*Return index 12 for the data struct*)
	13: getReal32 := data.ix13; (*Return index 13 for the data struct*)
	14: getReal32 := data.ix14; (*Return index 14 for the data struct*)
	15: getReal32 := data.ix15; (*Return index 15 for the data struct*)
	16: getReal32 := data.ix16; (*Return index 16 for the data struct*)
	17: getReal32 := data.ix17; (*Return index 17 for the data struct*)
	18: getReal32 := data.ix18; (*Return index 18 for the data struct*)
	19: getReal32 := data.ix19; (*Return index 19 for the data struct*)
	20: getReal32 := data.ix20; (*Return index 20 for the data struct*)
	21: getReal32 := data.ix21; (*Return index 21 for the data struct*)
	22: getReal32 := data.ix22; (*Return index 22 for the data struct*)
	23: getReal32 := data.ix23; (*Return index 23 for the data struct*)
	24: getReal32 := data.ix24; (*Return index 24 for the data struct*)
	25: getReal32 := data.ix25; (*Return index 25 for the data struct*)
	26: getReal32 := data.ix26; (*Return index 26 for the data struct*)
	27: getReal32 := data.ix27; (*Return index 27 for the data struct*)
	28: getReal32 := data.ix28; (*Return index 28 for the data struct*)
	29: getReal32 := data.ix29; (*Return index 29 for the data struct*)
	30: getReal32 := data.ix30; (*Return index 30 for the data struct*)
	31: getReal32 := data.ix31; (*Return index 31 for the data struct*)
ELSE
	(*Index is invalid, return initial function value*)
	RETURN;
END_CASE
RETURN;

          
END_FUNCTION

FUNCTION getSint32 : SINT
  VAR_INPUT
    data : SINT32;  (* Data to work on *)
    ix : USINT;  (* Index to retrieve *)
  END_VAR

            CASE ix OF
	0: getSint32 := data.ix00; (*Return index 0 for the data struct*)
	1: getSint32 := data.ix01; (*Return index 1 for the data struct*)
	2: getSint32 := data.ix02; (*Return index 2 for the data struct*)
	3: getSint32 := data.ix03; (*Return index 3 for the data struct*)
	4: getSint32 := data.ix04; (*Return index 4 for the data struct*)
	5: getSint32 := data.ix05; (*Return index 5 for the data struct*)
	6: getSint32 := data.ix06; (*Return index 6 for the data struct*)
	7: getSint32 := data.ix07; (*Return index 7 for the data struct*)
	8: getSint32 := data.ix08; (*Return index 8 for the data struct*)
	9: getSint32 := data.ix09; (*Return index 9 for the data struct*)
	10: getSint32 := data.ix10; (*Return index 10 for the data struct*)
	11: getSint32 := data.ix11; (*Return index 11 for the data struct*)
	12: getSint32 := data.ix12; (*Return index 12 for the data struct*)
	13: getSint32 := data.ix13; (*Return index 13 for the data struct*)
	14: getSint32 := data.ix14; (*Return index 14 for the data struct*)
	15: getSint32 := data.ix15; (*Return index 15 for the data struct*)
	16: getSint32 := data.ix16; (*Return index 16 for the data struct*)
	17: getSint32 := data.ix17; (*Return index 17 for the data struct*)
	18: getSint32 := data.ix18; (*Return index 18 for the data struct*)
	19: getSint32 := data.ix19; (*Return index 19 for the data struct*)
	20: getSint32 := data.ix20; (*Return index 20 for the data struct*)
	21: getSint32 := data.ix21; (*Return index 21 for the data struct*)
	22: getSint32 := data.ix22; (*Return index 22 for the data struct*)
	23: getSint32 := data.ix23; (*Return index 23 for the data struct*)
	24: getSint32 := data.ix24; (*Return index 24 for the data struct*)
	25: getSint32 := data.ix25; (*Return index 25 for the data struct*)
	26: getSint32 := data.ix26; (*Return index 26 for the data struct*)
	27: getSint32 := data.ix27; (*Return index 27 for the data struct*)
	28: getSint32 := data.ix28; (*Return index 28 for the data struct*)
	29: getSint32 := data.ix29; (*Return index 29 for the data struct*)
	30: getSint32 := data.ix30; (*Return index 30 for the data struct*)
	31: getSint32 := data.ix31; (*Return index 31 for the data struct*)
ELSE
	(*Index is invalid, return initial function value*)
	RETURN;
END_CASE
RETURN;

          
END_FUNCTION

FUNCTION getString32 : STRING
  VAR_INPUT
    data : STRING32;  (* Data to work on *)
    ix : USINT;  (* Index to retrieve *)
  END_VAR

            CASE ix OF
	0: getString32 := data.ix00; (*Return index 0 for the data struct*)
	1: getString32 := data.ix01; (*Return index 1 for the data struct*)
	2: getString32 := data.ix02; (*Return index 2 for the data struct*)
	3: getString32 := data.ix03; (*Return index 3 for the data struct*)
	4: getString32 := data.ix04; (*Return index 4 for the data struct*)
	5: getString32 := data.ix05; (*Return index 5 for the data struct*)
	6: getString32 := data.ix06; (*Return index 6 for the data struct*)
	7: getString32 := data.ix07; (*Return index 7 for the data struct*)
	8: getString32 := data.ix08; (*Return index 8 for the data struct*)
	9: getString32 := data.ix09; (*Return index 9 for the data struct*)
	10: getString32 := data.ix10; (*Return index 10 for the data struct*)
	11: getString32 := data.ix11; (*Return index 11 for the data struct*)
	12: getString32 := data.ix12; (*Return index 12 for the data struct*)
	13: getString32 := data.ix13; (*Return index 13 for the data struct*)
	14: getString32 := data.ix14; (*Return index 14 for the data struct*)
	15: getString32 := data.ix15; (*Return index 15 for the data struct*)
	16: getString32 := data.ix16; (*Return index 16 for the data struct*)
	17: getString32 := data.ix17; (*Return index 17 for the data struct*)
	18: getString32 := data.ix18; (*Return index 18 for the data struct*)
	19: getString32 := data.ix19; (*Return index 19 for the data struct*)
	20: getString32 := data.ix20; (*Return index 20 for the data struct*)
	21: getString32 := data.ix21; (*Return index 21 for the data struct*)
	22: getString32 := data.ix22; (*Return index 22 for the data struct*)
	23: getString32 := data.ix23; (*Return index 23 for the data struct*)
	24: getString32 := data.ix24; (*Return index 24 for the data struct*)
	25: getString32 := data.ix25; (*Return index 25 for the data struct*)
	26: getString32 := data.ix26; (*Return index 26 for the data struct*)
	27: getString32 := data.ix27; (*Return index 27 for the data struct*)
	28: getString32 := data.ix28; (*Return index 28 for the data struct*)
	29: getString32 := data.ix29; (*Return index 29 for the data struct*)
	30: getString32 := data.ix30; (*Return index 30 for the data struct*)
	31: getString32 := data.ix31; (*Return index 31 for the data struct*)
ELSE
	(*Index is invalid, return initial function value*)
	RETURN;
END_CASE
RETURN;

          
END_FUNCTION

FUNCTION getTime_of_day32 : TOD
  VAR_INPUT
    data : TIME_OF_DAY32;  (* Data to work on *)
    ix : USINT;  (* Index to retrieve *)
  END_VAR

            CASE ix OF
	0: getTime_of_day32 := data.ix00; (*Return index 0 for the data struct*)
	1: getTime_of_day32 := data.ix01; (*Return index 1 for the data struct*)
	2: getTime_of_day32 := data.ix02; (*Return index 2 for the data struct*)
	3: getTime_of_day32 := data.ix03; (*Return index 3 for the data struct*)
	4: getTime_of_day32 := data.ix04; (*Return index 4 for the data struct*)
	5: getTime_of_day32 := data.ix05; (*Return index 5 for the data struct*)
	6: getTime_of_day32 := data.ix06; (*Return index 6 for the data struct*)
	7: getTime_of_day32 := data.ix07; (*Return index 7 for the data struct*)
	8: getTime_of_day32 := data.ix08; (*Return index 8 for the data struct*)
	9: getTime_of_day32 := data.ix09; (*Return index 9 for the data struct*)
	10: getTime_of_day32 := data.ix10; (*Return index 10 for the data struct*)
	11: getTime_of_day32 := data.ix11; (*Return index 11 for the data struct*)
	12: getTime_of_day32 := data.ix12; (*Return index 12 for the data struct*)
	13: getTime_of_day32 := data.ix13; (*Return index 13 for the data struct*)
	14: getTime_of_day32 := data.ix14; (*Return index 14 for the data struct*)
	15: getTime_of_day32 := data.ix15; (*Return index 15 for the data struct*)
	16: getTime_of_day32 := data.ix16; (*Return index 16 for the data struct*)
	17: getTime_of_day32 := data.ix17; (*Return index 17 for the data struct*)
	18: getTime_of_day32 := data.ix18; (*Return index 18 for the data struct*)
	19: getTime_of_day32 := data.ix19; (*Return index 19 for the data struct*)
	20: getTime_of_day32 := data.ix20; (*Return index 20 for the data struct*)
	21: getTime_of_day32 := data.ix21; (*Return index 21 for the data struct*)
	22: getTime_of_day32 := data.ix22; (*Return index 22 for the data struct*)
	23: getTime_of_day32 := data.ix23; (*Return index 23 for the data struct*)
	24: getTime_of_day32 := data.ix24; (*Return index 24 for the data struct*)
	25: getTime_of_day32 := data.ix25; (*Return index 25 for the data struct*)
	26: getTime_of_day32 := data.ix26; (*Return index 26 for the data struct*)
	27: getTime_of_day32 := data.ix27; (*Return index 27 for the data struct*)
	28: getTime_of_day32 := data.ix28; (*Return index 28 for the data struct*)
	29: getTime_of_day32 := data.ix29; (*Return index 29 for the data struct*)
	30: getTime_of_day32 := data.ix30; (*Return index 30 for the data struct*)
	31: getTime_of_day32 := data.ix31; (*Return index 31 for the data struct*)
ELSE
	(*Index is invalid, return initial function value*)
	RETURN;
END_CASE
RETURN;

          
END_FUNCTION

FUNCTION getTime32 : TIME
  VAR_INPUT
    data : TIME32;  (* Data to work on *)
    ix : USINT;  (* Index to retrieve *)
  END_VAR

            CASE ix OF
	0: getTime32 := data.ix00; (*Return index 0 for the data struct*)
	1: getTime32 := data.ix01; (*Return index 1 for the data struct*)
	2: getTime32 := data.ix02; (*Return index 2 for the data struct*)
	3: getTime32 := data.ix03; (*Return index 3 for the data struct*)
	4: getTime32 := data.ix04; (*Return index 4 for the data struct*)
	5: getTime32 := data.ix05; (*Return index 5 for the data struct*)
	6: getTime32 := data.ix06; (*Return index 6 for the data struct*)
	7: getTime32 := data.ix07; (*Return index 7 for the data struct*)
	8: getTime32 := data.ix08; (*Return index 8 for the data struct*)
	9: getTime32 := data.ix09; (*Return index 9 for the data struct*)
	10: getTime32 := data.ix10; (*Return index 10 for the data struct*)
	11: getTime32 := data.ix11; (*Return index 11 for the data struct*)
	12: getTime32 := data.ix12; (*Return index 12 for the data struct*)
	13: getTime32 := data.ix13; (*Return index 13 for the data struct*)
	14: getTime32 := data.ix14; (*Return index 14 for the data struct*)
	15: getTime32 := data.ix15; (*Return index 15 for the data struct*)
	16: getTime32 := data.ix16; (*Return index 16 for the data struct*)
	17: getTime32 := data.ix17; (*Return index 17 for the data struct*)
	18: getTime32 := data.ix18; (*Return index 18 for the data struct*)
	19: getTime32 := data.ix19; (*Return index 19 for the data struct*)
	20: getTime32 := data.ix20; (*Return index 20 for the data struct*)
	21: getTime32 := data.ix21; (*Return index 21 for the data struct*)
	22: getTime32 := data.ix22; (*Return index 22 for the data struct*)
	23: getTime32 := data.ix23; (*Return index 23 for the data struct*)
	24: getTime32 := data.ix24; (*Return index 24 for the data struct*)
	25: getTime32 := data.ix25; (*Return index 25 for the data struct*)
	26: getTime32 := data.ix26; (*Return index 26 for the data struct*)
	27: getTime32 := data.ix27; (*Return index 27 for the data struct*)
	28: getTime32 := data.ix28; (*Return index 28 for the data struct*)
	29: getTime32 := data.ix29; (*Return index 29 for the data struct*)
	30: getTime32 := data.ix30; (*Return index 30 for the data struct*)
	31: getTime32 := data.ix31; (*Return index 31 for the data struct*)
ELSE
	(*Index is invalid, return initial function value*)
	RETURN;
END_CASE
RETURN;

          
END_FUNCTION

FUNCTION getUdint32 : UDINT
  VAR_INPUT
    data : UDINT32;  (* Data to work on *)
    ix : USINT;  (* Index to retrieve *)
  END_VAR

            CASE ix OF
	0: getUdint32 := data.ix00; (*Return index 0 for the data struct*)
	1: getUdint32 := data.ix01; (*Return index 1 for the data struct*)
	2: getUdint32 := data.ix02; (*Return index 2 for the data struct*)
	3: getUdint32 := data.ix03; (*Return index 3 for the data struct*)
	4: getUdint32 := data.ix04; (*Return index 4 for the data struct*)
	5: getUdint32 := data.ix05; (*Return index 5 for the data struct*)
	6: getUdint32 := data.ix06; (*Return index 6 for the data struct*)
	7: getUdint32 := data.ix07; (*Return index 7 for the data struct*)
	8: getUdint32 := data.ix08; (*Return index 8 for the data struct*)
	9: getUdint32 := data.ix09; (*Return index 9 for the data struct*)
	10: getUdint32 := data.ix10; (*Return index 10 for the data struct*)
	11: getUdint32 := data.ix11; (*Return index 11 for the data struct*)
	12: getUdint32 := data.ix12; (*Return index 12 for the data struct*)
	13: getUdint32 := data.ix13; (*Return index 13 for the data struct*)
	14: getUdint32 := data.ix14; (*Return index 14 for the data struct*)
	15: getUdint32 := data.ix15; (*Return index 15 for the data struct*)
	16: getUdint32 := data.ix16; (*Return index 16 for the data struct*)
	17: getUdint32 := data.ix17; (*Return index 17 for the data struct*)
	18: getUdint32 := data.ix18; (*Return index 18 for the data struct*)
	19: getUdint32 := data.ix19; (*Return index 19 for the data struct*)
	20: getUdint32 := data.ix20; (*Return index 20 for the data struct*)
	21: getUdint32 := data.ix21; (*Return index 21 for the data struct*)
	22: getUdint32 := data.ix22; (*Return index 22 for the data struct*)
	23: getUdint32 := data.ix23; (*Return index 23 for the data struct*)
	24: getUdint32 := data.ix24; (*Return index 24 for the data struct*)
	25: getUdint32 := data.ix25; (*Return index 25 for the data struct*)
	26: getUdint32 := data.ix26; (*Return index 26 for the data struct*)
	27: getUdint32 := data.ix27; (*Return index 27 for the data struct*)
	28: getUdint32 := data.ix28; (*Return index 28 for the data struct*)
	29: getUdint32 := data.ix29; (*Return index 29 for the data struct*)
	30: getUdint32 := data.ix30; (*Return index 30 for the data struct*)
	31: getUdint32 := data.ix31; (*Return index 31 for the data struct*)
ELSE
	(*Index is invalid, return initial function value*)
	RETURN;
END_CASE
RETURN;

          
END_FUNCTION

FUNCTION_BLOCK getUDT_Cmd32
  VAR_INPUT
    data : UDT_Cmd32;  (* Data to work on *)
    ix : USINT;  (* Index to retrieve *)
  END_VAR
  VAR_OUTPUT
    Out : UDT_Cmd;  (* Returned data *)
  END_VAR

            CASE ix OF
	0: Out := data.udt00; (*Return index 0 for the data struct*)
	1: Out := data.udt01; (*Return index 1 for the data struct*)
	2: Out := data.udt02; (*Return index 2 for the data struct*)
	3: Out := data.udt03; (*Return index 3 for the data struct*)
	4: Out := data.udt04; (*Return index 4 for the data struct*)
	5: Out := data.udt05; (*Return index 5 for the data struct*)
	6: Out := data.udt06; (*Return index 6 for the data struct*)
	7: Out := data.udt07; (*Return index 7 for the data struct*)
	8: Out := data.udt08; (*Return index 8 for the data struct*)
	9: Out := data.udt09; (*Return index 9 for the data struct*)
	10: Out := data.udt10; (*Return index 10 for the data struct*)
	11: Out := data.udt11; (*Return index 11 for the data struct*)
	12: Out := data.udt12; (*Return index 12 for the data struct*)
	13: Out := data.udt13; (*Return index 13 for the data struct*)
	14: Out := data.udt14; (*Return index 14 for the data struct*)
	15: Out := data.udt15; (*Return index 15 for the data struct*)
	16: Out := data.udt16; (*Return index 16 for the data struct*)
	17: Out := data.udt17; (*Return index 17 for the data struct*)
	18: Out := data.udt18; (*Return index 18 for the data struct*)
	19: Out := data.udt19; (*Return index 19 for the data struct*)
	20: Out := data.udt20; (*Return index 20 for the data struct*)
	21: Out := data.udt21; (*Return index 21 for the data struct*)
	22: Out := data.udt22; (*Return index 22 for the data struct*)
	23: Out := data.udt23; (*Return index 23 for the data struct*)
	24: Out := data.udt24; (*Return index 24 for the data struct*)
	25: Out := data.udt25; (*Return index 25 for the data struct*)
	26: Out := data.udt26; (*Return index 26 for the data struct*)
	27: Out := data.udt27; (*Return index 27 for the data struct*)
	28: Out := data.udt28; (*Return index 28 for the data struct*)
	29: Out := data.udt29; (*Return index 29 for the data struct*)
	30: Out := data.udt30; (*Return index 30 for the data struct*)
	31: Out := data.udt31; (*Return index 31 for the data struct*)
ELSE
	(*Index is invalid, return initial function value*)
	Out := Out;
END_CASE

          
END_FUNCTION_BLOCK

FUNCTION_BLOCK getUDT_Status32
  VAR_INPUT
    data : UDT_Status32;  (* Data to work on *)
    ix : USINT;  (* Index to retrieve *)
  END_VAR
  VAR_OUTPUT
    Out : UDT_Status;  (* Returned data *)
  END_VAR

            CASE ix OF
	0: Out := data.udt00; (*Return index 0 for the data struct*)
	1: Out := data.udt01; (*Return index 1 for the data struct*)
	2: Out := data.udt02; (*Return index 2 for the data struct*)
	3: Out := data.udt03; (*Return index 3 for the data struct*)
	4: Out := data.udt04; (*Return index 4 for the data struct*)
	5: Out := data.udt05; (*Return index 5 for the data struct*)
	6: Out := data.udt06; (*Return index 6 for the data struct*)
	7: Out := data.udt07; (*Return index 7 for the data struct*)
	8: Out := data.udt08; (*Return index 8 for the data struct*)
	9: Out := data.udt09; (*Return index 9 for the data struct*)
	10: Out := data.udt10; (*Return index 10 for the data struct*)
	11: Out := data.udt11; (*Return index 11 for the data struct*)
	12: Out := data.udt12; (*Return index 12 for the data struct*)
	13: Out := data.udt13; (*Return index 13 for the data struct*)
	14: Out := data.udt14; (*Return index 14 for the data struct*)
	15: Out := data.udt15; (*Return index 15 for the data struct*)
	16: Out := data.udt16; (*Return index 16 for the data struct*)
	17: Out := data.udt17; (*Return index 17 for the data struct*)
	18: Out := data.udt18; (*Return index 18 for the data struct*)
	19: Out := data.udt19; (*Return index 19 for the data struct*)
	20: Out := data.udt20; (*Return index 20 for the data struct*)
	21: Out := data.udt21; (*Return index 21 for the data struct*)
	22: Out := data.udt22; (*Return index 22 for the data struct*)
	23: Out := data.udt23; (*Return index 23 for the data struct*)
	24: Out := data.udt24; (*Return index 24 for the data struct*)
	25: Out := data.udt25; (*Return index 25 for the data struct*)
	26: Out := data.udt26; (*Return index 26 for the data struct*)
	27: Out := data.udt27; (*Return index 27 for the data struct*)
	28: Out := data.udt28; (*Return index 28 for the data struct*)
	29: Out := data.udt29; (*Return index 29 for the data struct*)
	30: Out := data.udt30; (*Return index 30 for the data struct*)
	31: Out := data.udt31; (*Return index 31 for the data struct*)
ELSE
	(*Index is invalid, return initial function value*)
	Out := Out;
END_CASE

          
END_FUNCTION_BLOCK

FUNCTION getUint32 : UINT
  VAR_INPUT
    data : UINT32;  (* Data to work on *)
    ix : USINT;  (* Index to retrieve *)
  END_VAR

